	//Init Zone		
	fbSortedListMoversInQueue.ListOfMoversToCheck := THIS^.fbAssignedMovers;
	fbSortedListMoversInQueue.AccocietedTrack := THIS^.AccocietedTrack;	
	
	bInitDone := TRUE;
ELSE
	//Done
	Initialize:= S_OK;
END_IF


THIS^.fbFeedback.ActiveCommand 		:= TO_STRING(CHALET_NC.E_NcAxisCommands.Initialize);
THIS^.eActiveCommand 				:= CHALET_NC.E_NcAxisCommands.Initialize;
THIS^.fbFeedback.LastCommandAccepted:= TRUE;	
//Set done or keep in busy state	
THIS^.fbFeedback.HR := Initialize;
END_METHOD

{attribute 'monitoring':='call'}
PROPERTY MoverGapAtExit : LREAL //[mm] Every mover that leaves or passes the station gets this new gap as a target.
GET
MoverGapAtExit := fMoverGapAtExit;
END_GET
SET
IF MoverGapAtExit < XPlanarParameterlist.F_MOVER_MINIMUM_GAP_ON_TRACK THEN
	MoverGapAtExit := XPlanarParameterlist.F_MOVER_MINIMUM_GAP_ON_TRACK;
END_IF

fMoverGapAtExit := MoverGapAtExit;
END_SET
END_PROPERTY

{attribute 'monitoring':='call'}
PROPERTY MoverVelocityAtExit : LREAL //[mm/s] Every mover that leaves or passes the station gets this new velocity as a target.
GET
MoverVelocityAtExit := fMoverVelocityAtExit;
END_GET
SET
fMoverVelocityAtExit := MoverVelocityAtExit;
END_SET
END_PROPERTY

{attribute 'monitoring':='call'}
PROPERTY PositionOnTrack : LREAL
GET
PositionOnTrack := THIS^.fPositionOnTrack;
END_GET
END_PROPERTY

{attribute 'monitoring':='call'}
PROPERTY PositionOnTrackXY : REFERENCE TO PositionXY
GET
PositionOnTrackXY REF= THIS^.fbPositionOnTrackXY;
END_GET
END_PROPERTY

{attribute 'monitoring':='call'}
PROPERTY PositionXY : REFERENCE TO  PositionXY
GET
PositionXY REF= THIS^.fbPositionPlanned;
END_GET
END_PROPERTY

METHOD RegistrateStationBehinde : HRESULT
VAR_INPUT
	ipStation : I_CH_Object;
END_VAR
VAR
	ipXpStation : I_XP_Station;
END_VAR
//Check if the input implements an station interface 
IF NOT ToXpStation(ipStation,ipXpStation) THEN
	RegistrateStationBehinde := E_FAIL;
	RETURN;
END_IF

//Check if not allready is added to list
IF THIS^.fbStationsBehinde.FindObject(ipStation) THEN
	;//Allready in List
ELSE	
	THIS^.fbStationsBehinde.AddObject(ipStation);
END_IF

RegistrateStationBehinde := S_OK;
END_METHOD

METHOD SearchNextBestStationByName : ST_PathFinder_1
VAR_INPUT
	sTargedStationGroupeID : STRING;
	nPermittedSearchDepth : UINT;
	ipWhoIsAsking	: I_XP_Station;

END_VAR
VAR
	nRemainingSearchDepth 			: UINT;
	ipThisStation 					: I_XP_Station;
	ipStation 						: I_XP_Station;
	stPath							: ST_PathFinder_1;
	bIamTheAsker					: BOOL;
	bTargetFoundOnThisPath			: BOOL;
	bStationIsOnlyForDynamicChanges : BOOL;
	bStationIsFull					: BOOL;
	bStationHanMoreMoverThanAllowed : BOOL;
	bStationHasAFreePlaceInQueue 	: BOOL;
	bStationIsNotReadyToRecvMovers	: BOOL;

END_VAR
ipThisStation := (THIS^);

//Invalide input
IF ipWhoIsAsking = 0 OR sTargedStationGroupeID = '' THEN
	searchNextBestStationByName.bTargetFound := FALSE;
	searchNextBestStationByName.ipBestStation := 0;
	RETURN;
END_IF

//Has the maximum search depth been reached?
nRemainingSearchDepth := nPermittedSearchDepth - 1;
IF nRemainingSearchDepth = 0 THEN
	searchNextBestStationByName.bTargetFound := FALSE;
	searchNextBestStationByName.ipBestStation := 0;
	RETURN;
END_IF

//Is the station not aware of any other stations in front of it?
IF THIS^.fbStationsAhead.Size = 0 THEN
	searchNextBestStationByName.bTargetFound := FALSE;
	searchNextBestStationByName.ipBestStation := 0;
	RETURN;
END_IF

//Check if the requested station is this one. And not the station who is searching
IF ((THIS^.StationGroupID = sTargedStationGroupeID) AND (ipWhoIsAsking <> ipThisStation)) THEN
	stPath.bTargetFound := TRUE;
	stPath.ipBestStation := THIS^;
ELSE
	//Check the stations ahead if a movement to targed station is posible. Multiple stations incase of an switch.
	THIS^.fbStationsAhead.ResetIterator();
	WHILE THIS^.fbStationsAhead.HasNextObject() DO
		IF ToXpStation(THIS^.fbStationsAhead.GetNextObject(),ipStation) THEN
			stPath := ipStation.searchNextBestStationByName(sTargedStationGroupeID, nRemainingSearchDepth, ipWhoIsAsking);
			//the information that we are on a valid path is set if a path to destination was detected
			IF stPath.bTargetFound THEN
				bTargetFoundOnThisPath := TRUE;
			END_IF
			//if a path is found with a valid in-between position, this should be used and the finder is aborted here
			IF stPath.ipBestStation <> 0 THEN
				EXIT;
			END_IF
		END_IF
	END_WHILE
	stPath.bTargetFound := bTargetFoundOnThisPath;
END_IF

//Abort - not a valide path
IF NOT stPath.bTargetFound THEN
	searchNextBestStationByName.bTargetFound := FALSE;
	searchNextBestStationByName.ipBestStation := 0;
	RETURN;
END_IF


//evaluate whether the current best station should be overwritten by this one
bIamTheAsker					:= ipWhoIsAsking = ipThisStation;
bStationHanMoreMoverThanAllowed := (THIS^.CtsMoversInQueue > THIS^.nMoverQueueSize); //Maybe during statup if all movers are forced to station x.	
bStationIsFull					:= (THIS^.CtsEmptySpaceInQueue = 0) AND NOT (THIS^.nMoverQueueSize = 0);
bStationHasAFreePlaceInQueue 	:= (THIS^.CtsEmptySpaceInQueue > 0);
bStationIsOnlyForDynamicChanges := (THIS^.nMoverQueueSize = 0);
//bStationIsTheTarged				:= (THIS^.StationGroupID = ipMover.TargedStation);
bStationIsNotReadyToRecvMovers	:= ( NOT THIS^.bReadyToRecvMovers); 

//End of search. Return found station
IF bIamTheAsker THEN
	searchNextBestStationByName.bTargetFound := stPath.bTargetFound;
	searchNextBestStationByName.ipBestStation := stPath.ipBestStation;


//Is THIS Station a "Dynamic change station" (Queuesize = 0) and has only the purpose tho change the gap of passing movers.
//in this case, the current path should be left as it is. the station is ignored,
ELSIF bStationIsOnlyForDynamicChanges THEN
	searchNextBestStationByName.bTargetFound := stPath.bTargetFound;
	searchNextBestStationByName.ipBestStation := stPath.ipBestStation;


//This station is full, no movement posible. Do not evaluate if this station is the asker.(Dont care if my own station is full atm.)
ELSIF bStationIsFull OR bStationHanMoreMoverThanAllowed OR bStationIsNotReadyToRecvMovers OR bStationIsOnlyForDynamicChanges THEN
	searchNextBestStationByName.bTargetFound := stPath.bTargetFound;
	searchNextBestStationByName.ipBestStation := 0;

	
//This station in an valide an good targed for the mover. return this station
	ELSE
	searchNextBestStationByName.bTargetFound := TRUE;
	searchNextBestStationByName.ipBestStation := (THIS^);
END_IF
END_METHOD

{attribute 'monitoring':='call'}
PROPERTY StationGroupID : STRING
GET
StationGroupID := THIS^.sStationGroupId;
END_GET
END_PROPERTY

{attribute 'monitoring':='call'}
PROPERTY StationsAhead : I_CH_List
GET
StationsAhead := THIS^.fbStationsAhead;
END_GET
END_PROPERTY

{attribute 'monitoring':='call'}
PROPERTY StationsBehinde : I_CH_List
GET
StationsBehinde := THIS^.fbStationsBehinde;
END_GET
END_PROPERTY

{attribute 'monitoring':='call'}
PROPERTY SuppressDynamicsChange : BOOL // Suppress to change the dynamic(Gap+velocity) of passing movers. This is usefull in startup
GET
SuppressDynamicsChange := bSuppressDynamicsChange;
END_GET
SET
bSuppressDynamicsChange := SuppressDynamicsChange;
END_SET
END_PROPERTY

METHOD Update : HRESULT
VAR
	ipFirstMoverInQueue: I_XP_Mover;
	ipFirstMoverInQueuePlc : I_XP_Mover_PLC;
	ipFirstMoverInQueueObj : I_CH_Object;
	iStation: I_XP_Station;
	stPath: ST_PathFinder_1;
	bValideStationToStartMove : BOOL;
	
	ipThisStation : I_XP_Station;
END_VAR
//Force to do init befor call update
IF NOT bInitDone THEN
	THIS^.Initialize();
	RETURN;
END_IF




// ********************** Set feedback depending on active command *******************************
IF THIS^.eActiveCommand <> E_NcAxisCommands.None THEN
	fbFeedback.ActiveCommand 	:= TO_STRING(THIS^.eActiveCommand);	
END_IF

CASE THIS^.eActiveCommand OF

	E_NcAxisCommands.Initialize:
		fbFeedback.Busy 			:= NOT THIS^.bInitDone;
		fbFeedback.Done 			:= THIS^.bInitDone;
		fbFeedback.ErrorId 			:= 0;
		                        	

	ELSE//External command in subclass
		;
END_CASE


// **********************  Stop to execute commands on .done or .error ***************************
IF fbFeedback.Done OR THIS^.fbFeedback.Error THEN
	eActiveCommand 				:= E_NcAxisCommands.None;
END_IF

// Process Simulation. All functionality packed into one method for easier overwriting
THIS^.Simulation();


// If enabled start station logic
IF THIS^.ipXpSystem.Enabled THEN

	//Detect mover who is passing the station whitout be in queue. Adjust to new Gap
	IF fbTrigger.MoverDetected AND (fbTrigger.MoverAtTrigger <> 0) AND NOT THIS^.bSuppressDynamicsChange THEN
		//Only if not in this queue
		ipThisStation := (THIS^);
		IF fbTrigger.MoverAtTrigger.ParentStation <> ipThisStation THEN
			fbTrigger.MoverAtTrigger.MoveOnTrack(ipTrack	:= fbTrigger.MoverAtTrigger.LastCmdTargedTrack,
												fPosition	:= fbTrigger.MoverAtTrigger.LastCmdTargedPosition, 
												fGap		:= THIS^.fMoverGapAtExit);
		END_IF
	END_IF	
	
	//Test if the first mover is in station and send him away, if the destination is not this station
	ipFirstMoverInQueuePlc := THIS^.MoversInQueue[0];
	IF (ipFirstMoverInQueuePlc <> 0) AND_THEN (ipFirstMoverInQueuePlc.TargetStationGroupID <> THIS^.StationGroupID) AND_THEN __QUERYINTERFACE(ipFirstMoverInQueuePlc,ipFirstMoverInQueue) THEN
		//Get a path
		stPath := THIS^.searchNextBestStationByName(sTargedStationGroupeID := ipFirstMoverInQueue.TargetStationGroupID, nPermittedSearchDepth := XPlanarParameterlist.N_MAX_SEARCH_DEPTH, ipWhoIsAsking := (THIS^));
		bValideStationToStartMove := stPath.bTargetFound AND (stPath.ipBestStation <> 0);
		//Start Movement
		IF bValideStationToStartMove THEN 
			//deregister from this station and register with a new parrent station
			ipFirstMoverInQueueObj := THIS^.fbAssignedMovers.FindOID(ipFirstMoverInQueue.OID);
			THIS^.fbAssignedMovers.RemoveObject(ipFirstMoverInQueueObj);
			stPath.ipBestStation.AddMoverToQueue(ipFirstMoverInQueue);	

			//If mover is standstill in current station, send him away whit the exit gap, else use the in mover stored gap
			IF LREAL_TO_DINT(ipFirstMoverInQueue.PositionOnTrack) = LREAL_TO_DINT(THIS^.PositionOnTrack) THEN
				ipFirstMoverInQueue.MoveOnTrackToStation(ipStation := stPath.ipBestStation,
											fGap:= THIS^.fMoverGapAtExit);					
			ELSE
				ipFirstMoverInQueue.MoveOnTrackToStation(ipStation := stPath.ipBestStation,
								fGap:= ipFirstMoverInQueue.LastCmdTargedGap);
	
			END_IF	
 		END_IF     
	END_IF
END_IF



Update := S_OK;
END_METHOD

END_FUNCTION_BLOCK

// COMPONENTs/Stationen/I_XP_Station_PLC
INTERFACE I_XP_Station_PLC EXTENDS __SYSTEM.IQueryInterface

{attribute 'monitoring':='call'}
PROPERTY AreMoversInPlace : BOOL
GET
END_GET
END_PROPERTY

{attribute 'monitoring':='call'}
PROPERTY CtsEmptySpaceInQueue : UDINT
GET
END_GET
END_PROPERTY

{attribute 'monitoring':='call'}
PROPERTY CtsMoversInQueue : UDINT
GET
END_GET
END_PROPERTY

{attribute 'monitoring':='call'}
(* Return interface to mover in station. Return 0 if no mover is in station *)
PROPERTY InterfaceToMover : I_XP_Mover
GET
END_GET
END_PROPERTY

{attribute 'monitoring':='call'}
PROPERTY MoverQueueSize : UINT
GET
END_GET
SET
END_SET
END_PROPERTY

{attribute 'monitoring':='call'}
PROPERTY MoversInQueue : REFERENCE TO ARRAY [0..(CHALET_BaseComponents.BaseParameterlist.MAX_OBJECTS-1)] OF I_XP_Mover_PLC // Return a sorted list of movers in this zone. Index 0 is the mover in Front
GET
END_GET
END_PROPERTY

{attribute 'monitoring':='call'}
//prevent further movers from entering the station, 
//e.g. to prevent a collision. All movers that are already moving to reach this station will be stopped with a stop 
//and restarted with Ready True.
PROPERTY ReadyToRecvMovers : BOOL
GET
END_GET
SET
END_SET
END_PROPERTY

METHOD SendMoversToGroup : I_CH_Feedback
VAR_INPUT 
	sTargetStationGroupID : STRING;
END_VAR
END_METHOD

{attribute 'monitoring':='call'}
PROPERTY TargetPosMonitoringTime : TIME
GET
END_GET
SET
END_SET
END_PROPERTY

{attribute 'monitoring':='call'}
PROPERTY TargetPosWindow : LREAL
GET
END_GET
SET
END_SET
END_PROPERTY

{attribute 'monitoring':='call'}
PROPERTY ProcessSimulationActive : BOOL
GET
END_GET
END_PROPERTY

//If a valid time (>0seconds) is set and the configured destination station exists, then the movers will be sent away automatically after this time from now on.
METHOD SimulationMode : HRESULT
VAR_INPUT
	fProcessDuration 			: LREAL; //[s]
	sTargedStationGroupID		: STRING; //group of the targed station to automatic send after the duration
END_VAR
END_METHOD

{attribute 'monitoring':='call'}
PROPERTY AccocietedTrack : I_XP_Track
GET
END_GET
END_PROPERTY

{attribute 'monitoring':='call'}
PROPERTY Feedback : I_CH_Feedback
GET
END_GET
END_PROPERTY

{attribute 'monitoring':='call'}
PROPERTY MoverGapAtExit : LREAL //[mm] Every mover that leaves or passes the station gets this new gap as a target.
GET
END_GET
SET
END_SET
END_PROPERTY

{attribute 'monitoring':='call'}
PROPERTY PositionOnTrack : LREAL
GET
END_GET
END_PROPERTY

{attribute 'monitoring':='call'}
PROPERTY PositionOnTrackXY : REFERENCE TO PositionXY
GET
END_GET
END_PROPERTY

{attribute 'monitoring':='call'}
PROPERTY PositionXY : REFERENCE TO  PositionXY
GET
END_GET
END_PROPERTY

{attribute 'monitoring':='call'}
PROPERTY StationGroupID : STRING
GET
END_GET
END_PROPERTY

{attribute 'monitoring':='call'}
PROPERTY StationsAhead : I_CH_List
GET
END_GET
END_PROPERTY

{attribute 'monitoring':='call'}
PROPERTY StationsBehinde : I_CH_List
GET
END_GET
END_PROPERTY

END_INTERFACE

// COMPONENTs/Trigger/FB_XP_Trigger
{attribute 'no_explicit_call' := 'Do not call the body - Stick to OOP'}
FUNCTION_BLOCK FB_XP_Trigger EXTENDS FB_CH_Object IMPLEMENTS I_XP_Trigger
VAR
	{attribute 'hide'}
	bInitDone : BOOL;
	{attribute 'hide'}
	ipXpSystem : I_XP_System_Registration;
	{attribute 'hide'}
	ipAccocietedTrack : I_XP_Track;
	{attribute 'hide'}
	ipListOfMoversToCheck : CHALET_BaseComponents.I_CH_LIST;
	{attribute 'hide'}
	fTriggerPositionOnTrack : LREAL;
	{attribute 'hide'}
	eTriggerDirection : Tc3_Mc3Definitions.MC_Direction := Tc3_Mc3Definitions.MC_DIRECTION.mcDirectionPositive;
	{attribute 'hide'}
	ipMoverAtTrigger : I_XP_Mover;
	{attribute 'hide'}
	aMoversPositionLastCycle : ARRAY [0..(CHALET_BaseComponents.BaseParameterlist.MAX_OBJECTS-1)] OF LREAL; // This list is generated at the end of the PRG and contais the positions. The positions are checked in the next cycle
	{attribute 'hide'}
	aMoversTrackLastCycle : ARRAY [0..(CHALET_BaseComponents.BaseParameterlist.MAX_OBJECTS-1)] OF I_XP_Track; // This list is generated at the end of the PRG and contais the track. The tracks are checked in the next cycle
	{attribute 'hide'}
	aMoversInterfaceLastCycle : ARRAY [0..(CHALET_BaseComponents.BaseParameterlist.MAX_OBJECTS-1)] OF I_XP_Mover; // This list is generated at the end of the PRG and contais the Mover interface. The positions are checked in the next cycle
END_VAR

{attribute 'monitoring':='call'}
PROPERTY AccocietedTrack : I_XP_Track
GET
AccocietedTrack := THIS^.ipAccocietedTrack;
END_GET
SET
THIS^.ipAccocietedTrack := AccocietedTrack;
END_SET
END_PROPERTY

METHOD FB_init : BOOL
VAR_INPUT
	bInitRetains : BOOL; // if TRUE, the retain variables are initialized (warm start / cold start)
	bInCopyCode : BOOL;  // if TRUE, the instance afterwards gets moved into the copy code (online change)
	
	ipXpSystem : I_XP_System_Registration; //Interface to XTS system object
	
END_VAR
VAR_INST
	{attribute 'hide'}
	bFBInitCalledOnce : BOOL; //Do the following code once during start up and not during onlinechange
END_VAR
//Do the following code once during start up and not during onlinechange
IF NOT bFBInitCalledOnce THEN 
	;
END_IF

//Regristrate object in System if unknown
IF ipXpSystem <> 0 AND THIS^.ipXpSystem = 0 THEN
	ipXpSystem.RegisterTrigger(THIS^);
	THIS^.ipXpSystem := ipXpSystem;
END_IF

bFBInitCalledOnce := TRUE;
END_METHOD

{attribute 'monitoring':='call'}
PROPERTY HR : HRESULT
GET
IF ipAccocietedTrack <> 0 AND_THEN ipAccocietedTrack.Length > 0 THEN
	HR := S_OK;
ELSE
	HR := E_FAIL;
END_IF
END_GET
END_PROPERTY

METHOD Initialize : HRESULT
IF THIS^.ipXpSystem = 0 THEN
	//No valide interface
	Initialize := E_FAIL;
	RETURN;
END_IF

IF (THIS^.ipListOfMoversToCheck <> 0) AND (THIS^.ipAccocietedTrack <> 0) THEN
	THIS^.bInitDone := TRUE;
	Initialize := S_OK;
ELSE
	Initialize := E_FAIL;
END_IF
END_METHOD

PROPERTY ListOfMoversToCheck : I_CH_List
SET
IF ListOfMoversToCheck <> 0 THEN
	ipListOfMoversToCheck := ListOfMoversToCheck;
END_IF
END_SET
END_PROPERTY

{attribute 'monitoring':='call'}
PROPERTY MoverAtTrigger : I_XP_Mover
GET
THIS^.Prepare();//Prepare Time-critical information

MoverAtTrigger := ipMoverAtTrigger;
END_GET
END_PROPERTY

{attribute 'monitoring':='call'}
PROPERTY MoverDetected : BOOL
GET
THIS^.Prepare();//Prepare Time-critical information

MoverDetected := (ipMoverAtTrigger <> 0);
END_GET
END_PROPERTY

{attribute 'monitoring':='call'}
PROPERTY PositionOnTrack : LREAL
GET
PositionOnTrack := fTriggerPositionOnTrack;
END_GET
SET
fTriggerPositionOnTrack := PositionOnTrack;
END_SET
END_PROPERTY

(* Time-critical information is processed here, which can then be polled via the property every cycle. 
The update method is usually at the end of the program and then it is already 'outdated'. *)
METHOD PRIVATE Prepare : HRESULT
VAR
	fTrackLentgh : LREAL;
	fMoverActPos,fMoverLastPos : LREAL;
	ipMoverActTrack, ipMoverLastTrack : I_XP_Track;
	fRangePositive, fRangeNegative : LREAL;
	bTriggerIsCloseAtStartTrack, bTriggerIsCloseAtEndTrack : BOOL;
	bMoverWasInRangeNeg, bMoverWasInRangePos, bMoverIsInRangeNeg, bMoverIsInRangePos : BOOL;
	bMoverIsOnSameTrack, bMoverIsOnTrackAhead, bMoverIsOnTrackBehind, bMoverWasOnTrackAhead, bMoverWasOnTrackBehind : BOOL;
	nIdx, nIdxTrack : UDINT;
	fMaxMoveDistPerCycle : LREAL; //[mm] (2 m/s(max. xPlanar speed) * 20ms(max realistic SPS cycle time) + 10%)
END_VAR
VAR_INST
	{attribute 'hide'}
	nLastUpdatedCycleCount : UDINT;
END_VAR
VAR CONSTANT
END_VAR
//Check if this Cycle the dates are allready prepared
IF nLastUpdatedCycleCount <> TwinCAT_SystemInfoVarList._TaskInfo[THIS^.nTaskIndex].CycleCount THEN
	nLastUpdatedCycleCount := TwinCAT_SystemInfoVarList._TaskInfo[THIS^.nTaskIndex].CycleCount;
	
	//Abort on invalide interface - Get Track length
	IF ipAccocietedTrack = 0 THEN
		RETURN;
	END_IF
	fTrackLentgh := ipAccocietedTrack.Length;
	
	//Maximum distance a mover can travel in 1 plc cycle. Worstcase 2 m/s(max. xPlanar speed) * 20ms(max realistic SPS cycle time) + 10%
	fMaxMoveDistPerCycle := 2000.0(*2000mm/s=2mm/ms*) * (TwinCAT_SystemInfoVarList._TaskInfo[THIS^.nTaskIndex].CycleTime(*[100ns]*)/10_000)(*CycleTime ms*) / 1000.0 * 1.1(*10%*);
	
	//Clear last stored Mover if an new cycle has started
	THIS^.ipMoverAtTrigger := 0;
	
	//Check old list of Moverspositions and compare them to the current position of the same mover.
	//Set Trigger if the Mover pass the Station
	fRangePositive := MIN((THIS^.fTriggerPositionOnTrack + fMaxMoveDistPerCycle),fTrackLentgh);
	fRangeNegative := MAX((THIS^.fTriggerPositionOnTrack - fMaxMoveDistPerCycle),0); 
	bTriggerIsCloseAtStartTrack := (THIS^.fTriggerPositionOnTrack - fMaxMoveDistPerCycle) < 0.0;
	bTriggerIsCloseAtEndTrack 	:= (THIS^.fTriggerPositionOnTrack + fMaxMoveDistPerCycle) > fTrackLentgh;

		
	FOR nIdx := 0 TO (CHALET_BaseComponents.BaseParameterlist.MAX_OBJECTS-1) DO
		
		IF aMoversInterfaceLastCycle[nIdx] <> 0 THEN
			fMoverActPos 			:= aMoversInterfaceLastCycle[nIdx].PositionOnTrack;
			fMoverLastPos			:= aMoversPositionLastCycle[nIdx];
			ipMoverActTrack 		:= aMoversInterfaceLastCycle[nIdx].CurrentTrack;
			ipMoverLastTrack 		:= aMoversTrackLastCycle[nIdx];
			bMoverIsOnSameTrack 	:= (ipMoverActTrack = ipAccocietedTrack);
			
			//Abort if Lasttrack is not known. Example: first cycle after enabling
			IF ipMoverActTrack = 0 OR ipMoverLastTrack = 0 THEN
				RETURN;
			END_IF
			
			//Reset flags 
			bMoverIsOnTrackAhead 	:= FALSE;		bMoverIsOnTrackBehind 	:= FALSE;		bMoverWasOnTrackAhead 	:= FALSE;		bMoverWasOnTrackBehind 	:= FALSE;
			
			//Test all tracks before and after this track to recognize that the mover has just changed tracks. 
			//This is important if this trigger is near the end or beginning of a track
			FOR nIdxTrack := 0 TO (XPlanarParameterlist.N_MAX_STATIONS_AHEAD_OR_BEHIND-1) DO
				//Tracks Ahead - Mover Is/Was on Track ahead and close(cMaxMoveDistPerCycle) at beginn on track
				IF ipMoverActTrack.TracksStartFromThis[nIdxTrack] <> 0 THEN
					bMoverIsOnTrackAhead 	:= bMoverIsOnTrackAhead 	OR ((ipAccocietedTrack = ipMoverActTrack.TracksStartFromThis[nIdxTrack])  AND ((fMoverActPos - fMaxMoveDistPerCycle) < 0.0));
					bMoverWasOnTrackAhead 	:= bMoverWasOnTrackAhead 	OR ((ipAccocietedTrack = ipMoverLastTrack.TracksStartFromThis[nIdxTrack]) AND ((fMoverLastPos - fMaxMoveDistPerCycle) < 0.0));
				END_IF
				//Tracks Behind - Mover Is/Was on Track behind and close(cMaxMoveDistPerCycle) at end on track
				IF ipMoverActTrack.TracksEndAtThis[nIdxTrack] <> 0 THEN
					bMoverIsOnTrackBehind 	:= bMoverIsOnTrackBehind 	OR ((ipAccocietedTrack = ipMoverActTrack.TracksEndAtThis[nIdxTrack])  AND ((fMoverActPos	+ fMaxMoveDistPerCycle) > ipMoverActTrack.Length));
					bMoverWasOnTrackBehind 	:= bMoverWasOnTrackBehind 	OR ((ipAccocietedTrack = ipMoverLastTrack.TracksEndAtThis[nIdxTrack]) AND ((fMoverLastPos 	+ fMaxMoveDistPerCycle) > ipMoverLastTrack.Length));
				END_IF
			END_FOR
			
			//Closed track and station in close to Modulo pos
			IF bMoverIsOnSameTrack THEN
				bMoverIsOnTrackAhead 	:= ((fMoverActPos - fMaxMoveDistPerCycle) < 0.0);
				bMoverWasOnTrackAhead 	:= ((fMoverLastPos - fMaxMoveDistPerCycle) < 0.0);
				bMoverIsOnTrackBehind 	:= ((fMoverActPos	+ fMaxMoveDistPerCycle) > ipMoverActTrack.Length);
				bMoverWasOnTrackBehind 	:= ((fMoverLastPos 	+ fMaxMoveDistPerCycle) > ipMoverLastTrack.Length);
			END_IF
			
			//Check if Mover passes the station. Ex.: If the Trigger is at Pos 0mm on track, the Mover is never in bRangeNeg. For this case check for bMoverOnTrackBefore
			bMoverIsInRangePos 		:= ((fMoverActPos >= THIS^.fTriggerPositionOnTrack) AND (fMoverActPos <= fRangePositive) AND bMoverIsOnSameTrack) OR (bMoverIsOnTrackAhead 	 AND bTriggerIsCloseAtEndTrack);   
			bMoverIsInRangeNeg 		:= ((fMoverActPos <= THIS^.fTriggerPositionOnTrack) AND (fMoverActPos >= fRangeNegative) AND bMoverIsOnSameTrack) OR (bMoverIsOnTrackBehind  AND bTriggerIsCloseAtStartTrack);     
			bMoverWasInRangePos		:= ((fMoverLastPos > THIS^.fTriggerPositionOnTrack) AND (fMoverLastPos >= fRangeNegative) AND bMoverIsOnSameTrack) OR (bMoverWasOnTrackAhead  AND bTriggerIsCloseAtEndTrack);   
			bMoverWasInRangeNeg		:= ((fMoverLastPos < THIS^.fTriggerPositionOnTrack) AND (fMoverLastPos <= fRangePositive) AND bMoverIsOnSameTrack) OR (bMoverWasOnTrackBehind AND bTriggerIsCloseAtStartTrack);     			

			IF eTriggerDirection = Tc3_Mc3Definitions.MC_DIRECTION.mcDirectionPositive  AND bMoverWasInRangeNeg AND bMoverIsInRangePos AND NOT bMoverWasInRangePos THEN
				THIS^.ipMoverAtTrigger := aMoversInterfaceLastCycle[nIdx];
				RETURN;
			ELSIF eTriggerDirection = Tc3_Mc3Definitions.MC_DIRECTION.mcDirectionNegative AND bMoverIsInRangeNeg AND bMoverWasInRangePos AND NOT bMoverWasInRangeNeg THEN
				THIS^.ipMoverAtTrigger := aMoversInterfaceLastCycle[nIdx];
				RETURN;	
			END_IF
			
		END_IF
	END_FOR
END_IF
END_METHOD

{attribute 'monitoring':='call'}
PROPERTY TimeStamp : Tc2_EtherCAT.T_DCTIME64
GET
THIS^.Prepare();//Prepare Time-critical information

///zzz todo exact time stamp calculatioin
 IF ipMoverAtTrigger <> 0 THEN
	 TimeStamp := F_GetCurDcTaskTime64();
 ELSE
	 TimeStamp := 0;
 END_IF
END_GET
END_PROPERTY

{attribute 'monitoring':='call'}
PROPERTY TriggerDirection : Tc3_Mc3Definitions.MC_Direction
GET
TriggerDirection := eTriggerDirection;
END_GET
SET
IF TriggerDirection =Tc3_Mc3Definitions.MC_DIRECTION.mcDirectionPositive OR TriggerDirection = Tc3_Mc3Definitions.MC_DIRECTION.mcDirectionNegative THEN
	eTriggerDirection := TriggerDirection;
END_IF
END_SET
END_PROPERTY

METHOD Update : HRESULT
VAR
	nIndex : UINT;
	ipMover : I_XP_Mover;
END_VAR
//Force to do an init befor call update
IF NOT bInitDone THEN
	THIS^.Initialize();
	RETURN;
END_IF

//Clear array
MEMSET(destAddr:=ADR(aMoversInterfaceLastCycle),n:=SIZEOF(aMoversInterfaceLastCycle),fillByte:=0);
MEMSET(destAddr:=ADR(aMoversPositionLastCycle),n:=SIZEOF(aMoversPositionLastCycle),fillByte:=0);
MEMSET(destAddr:=ADR(aMoversTrackLastCycle),n:=SIZEOF(aMoversTrackLastCycle),fillByte:=0);

nIndex := 0;
THIS^.ipListOfMoversToCheck.ResetIterator();
WHILE THIS^.ipListOfMoversToCheck.HasNextObject() DO
	
	//Cheack all Movers fill the actposition in the array
	IF ToXpMover(THIS^.ipListOfMoversToCheck.GetNextObject(),ipMover) THEN
		aMoversInterfaceLastCycle[nIndex] 	:= ipMover;
		aMoversPositionLastCycle[nIndex] 	:= ipMover.PositionOnTrack;
		aMoversTrackLastCycle[nIndex]		:= ipMover.CurrentTrack;
		nIndex := nIndex +1;
	END_IF
	
END_WHILE
END_METHOD

END_FUNCTION_BLOCK

// COMPONENTs/Trigger/I_XP_Trigger
INTERFACE I_XP_Trigger  EXTENDS __SYSTEM.IQueryInterface

{attribute 'monitoring':='call'}
PROPERTY AccocietedTrack : I_XP_Track
GET
END_GET
SET
END_SET
END_PROPERTY

{attribute 'monitoring':='call'}
PROPERTY HR : HRESULT
GET
END_GET
END_PROPERTY

PROPERTY ListOfMoversToCheck : I_CH_List
SET
END_SET
END_PROPERTY

{attribute 'monitoring':='call'}
PROPERTY MoverAtTrigger : I_XP_Mover
GET
END_GET
END_PROPERTY

{attribute 'monitoring':='call'}
PROPERTY MoverDetected : BOOL
GET
END_GET
END_PROPERTY

{attribute 'monitoring':='call'}
PROPERTY PositionOnTrack : LREAL
GET
END_GET
SET
END_SET
END_PROPERTY

{attribute 'monitoring':='call'}
PROPERTY TimeStamp : T_DCTIME64;
GET
END_GET
END_PROPERTY

{attribute 'monitoring':='call'}
PROPERTY TriggerDirection : Tc3_Mc3Definitions.MC_Direction
GET
END_GET
SET
END_SET
END_PROPERTY

END_INTERFACE

// COMPONENTs/Zone/FB_XP_Zone
{attribute 'no_explicit_call' := 'Do not call the body - Stick to OOP'}
// Check zone start to end in positive direktion.
FUNCTION_BLOCK FB_XP_Zone EXTENDS FB_CH_Object IMPLEMENTS I_XP_Zone
VAR
	{attribute 'hide'}
	bInitDone : BOOL;
	{attribute 'hide'}
	ipXpSystem : I_XP_System_Registration; //Interface to XPlanar system 
	{attribute 'hide'}
	ipListOfMoversToCheck : CHALET_BaseComponents.I_CH_LIST;
	{attribute 'hide'}
	aMoversInZone : ARRAY [0..(CHALET_BaseComponents.BaseParameterlist.MAX_OBJECTS-1)] OF I_XP_Mover_PLC;
	{attribute 'hide'}
	fStartPositionOnTrack : LREAL;
	{attribute 'hide'}
	fEndPositionOnTrack : LREAL;	
	{attribute 'hide'}
	ipAccocietedTrack : I_XP_Track;
END_VAR

{attribute 'monitoring':='call'}
PROPERTY AccocietedTrack : I_XP_Track
GET
AccocietedTrack := THIS^.ipAccocietedTrack;
END_GET
SET
THIS^.ipAccocietedTrack := AccocietedTrack;
END_SET
END_PROPERTY

{attribute 'monitoring':='call'}
PROPERTY CtsMoversInZone : UINT
GET
VAR
	nIndex : UDINT;
END_VAR
THIS^.Prepare();//Prepare Time-critical information

//Check array for entrys, exit if fisrt empty arrayindex is found.
FOR nIndex := 0 TO (CHALET_BaseComponents.BaseParameterlist.MAX_OBJECTS-1) DO
	IF (aMoversInZone[nIndex] <> 0) THEN
		CtsMoversInZone := CtsMoversInZone +1;
	ELSE
		RETURN;
	END_IF
END_FOR
END_GET
END_PROPERTY

{attribute 'monitoring':='call'}
PROPERTY EndPositionOnTrack : LREAL
GET
EndPositionOnTrack := fEndPositionOnTrack;
END_GET
SET
fEndPositionOnTrack := EndPositionOnTrack;
END_SET
END_PROPERTY

METHOD FB_init : BOOL
VAR_INPUT
	bInitRetains : BOOL; // if TRUE, the retain variables are initialized (warm start / cold start)
	bInCopyCode : BOOL;  // if TRUE, the instance afterwards gets moved into the copy code (online change)
	
	ipXpSystem : I_XP_System_Registration; //Interface to XPlanar system object
END_VAR
VAR_INST
	{attribute 'hide'}
	bFBInitCalledOnce : BOOL; //Do the following code once during start up and not during onlinechange
END_VAR
//Do the following code once during start up and not during onlinechange
IF NOT bFBInitCalledOnce THEN 
	;
END_IF

//Regristrate object in System if unknown
IF ipXpSystem <> 0 AND THIS^.ipXpSystem = 0 THEN
	ipXpSystem.RegisterZone(THIS^);
	THIS^.ipXpSystem := ipXpSystem;
END_IF

bFBInitCalledOnce := TRUE;
END_METHOD

{attribute 'monitoring':='call'}
PROPERTY HR : HRESULT
GET
IF ipAccocietedTrack <> 0 AND_THEN ipAccocietedTrack.Length > 0 THEN
	HR := S_OK;
ELSE
	HR := E_FAIL;
END_IF
END_GET
END_PROPERTY

METHOD Initialize : HRESULT
IF THIS^.ipXpSystem = 0 THEN
	//No valide interface
	Initialize := E_FAIL;
	RETURN;
END_IF


IF (THIS^.ipListOfMoversToCheck <> 0) AND (THIS^.ipAccocietedTrack <> 0) THEN
	THIS^.bInitDone := TRUE;
	Initialize := S_OK;
ELSE
	Initialize := E_FAIL;
END_IF
END_METHOD

PROPERTY ListOfMoversToCheck : I_CH_List
SET
IF ListOfMoversToCheck <> 0 THEN
	ipListOfMoversToCheck := ListOfMoversToCheck;
END_IF
END_SET
END_PROPERTY

{attribute 'monitoring':='call'}
PROPERTY MoversInZone : REFERENCE TO ARRAY [0..(CHALET_BaseComponents.BaseParameterlist.MAX_OBJECTS-1)] OF I_XP_Mover_PLC // Return a sorted list of movers in this zone. Index 0 is the mover in Front.
GET
THIS^.Prepare();//Prepare Time-critical information

MoversInZone REF= THIS^.aMoversInZone;
END_GET
END_PROPERTY

(* Time-critical information is processed here, which can then be polled via the property every cycle. 
The update method is usually at the end of the program and then it is already 'outdated'. *)
METHOD PRIVATE Prepare : HRESULT
VAR
	nLoopIndex : UDINT;
	ipMoverPlc : I_XP_Mover_PLC;
	fDistToStart : LREAL;
	aDisanceToStart : ARRAY [0..(CHALET_BaseComponents.BaseParameterlist.MAX_OBJECTS-1)] OF LREAL;
END_VAR
VAR_INST
	{attribute 'hide'}
	nLastUpdatedCycleCount : UDINT;
END_VAR
//Check if this Cycle the dates are allready prepared
IF nLastUpdatedCycleCount <> TwinCAT_SystemInfoVarList._TaskInfo[THIS^.nTaskIndex].CycleCount THEN
	nLastUpdatedCycleCount := TwinCAT_SystemInfoVarList._TaskInfo[THIS^.nTaskIndex].CycleCount;

	//Clear array
	MEMSET(destAddr:=ADR(aMoversInZone),n:=SIZEOF(aMoversInZone),fillByte:=0);
	
	//Cheack all Movers and generate a sorted list of all mover in this zone
	THIS^.ipListOfMoversToCheck.ResetIterator();
	WHILE THIS^.ipListOfMoversToCheck.HasNextObject() DO
		IF __QUERYINTERFACE(THIS^.ipListOfMoversToCheck.GetNextObject(),ipMoverPlc) THEN
			
			//If in zone
			IF ipMoverPlc.CurrentTrack = THIS^.ipAccocietedTrack AND_THEN (fStartPositionOnTrack <= ipMoverPlc.PositionOnTrack) AND (fEndPositionOnTrack >= ipMoverPlc.PositionOnTrack) AND (fStartPositionOnTrack <= fEndPositionOnTrack) THEN
				fDistToStart := fEndPositionOnTrack - ipMoverPlc.PositionOnTrack;
				
				//Check array of movers and decide if the current one is closer to 
				FOR nLoopIndex := 0 TO (CHALET_BaseComponents.BaseParameterlist.MAX_OBJECTS-1) DO
					//empty array position
					IF aMoversInZone[nLoopIndex] = 0 THEN
						aMoversInZone[nLoopIndex] := ipMoverPlc;
						aDisanceToStart[nLoopIndex] := fDistToStart;
						EXIT;
						
					//Closer Mover found, move whole array 	
					ELSIF aDisanceToStart[nLoopIndex] > fDistToStart THEN
						MEMMOVE(srcAddr := ADR(aMoversInZone[nLoopIndex]), destAddr := ADR(aMoversInZone[nLoopIndex+1]), n := (SIZEOF(aMoversInZone[0])*(CHALET_BaseComponents.BaseParameterlist.MAX_OBJECTS-1)));
						MEMMOVE(srcAddr := ADR(aDisanceToStart[nLoopIndex]), destAddr := ADR(aDisanceToStart[nLoopIndex+1]), n := (SIZEOF(aDisanceToStart[0])*(CHALET_BaseComponents.BaseParameterlist.MAX_OBJECTS-1)));
						aMoversInZone[nLoopIndex] := ipMoverPlc;
						aDisanceToStart[nLoopIndex] := fDistToStart;
						EXIT;
						
					//check next position	
					ELSE 
						;
					END_IF
				END_FOR
			END_IF
		END_IF
	END_WHILE
END_IF
END_METHOD

{attribute 'monitoring':='call'}
PROPERTY StartPositionOnTrack : LREAL
GET
StartPositionOnTrack := fStartPositionOnTrack;
END_GET
SET
fStartPositionOnTrack := StartPositionOnTrack;
END_SET
END_PROPERTY

METHOD Update : HRESULT
VAR

END_VAR
// Nothing todo in Update. Check Prepare
END_METHOD

END_FUNCTION_BLOCK

// COMPONENTs/Zone/I_XP_Zone
INTERFACE I_XP_Zone

{attribute 'monitoring':='call'}
PROPERTY AccocietedTrack : I_XP_Track
GET
END_GET
SET
END_SET
END_PROPERTY

{attribute 'monitoring':='call'}
PROPERTY CtsMoversInZone : UINT
GET
END_GET
END_PROPERTY

{attribute 'monitoring':='call'}
PROPERTY EndPositionOnTrack : LREAL
GET
END_GET
SET
END_SET
END_PROPERTY

{attribute 'monitoring':='call'}
PROPERTY HR : HRESULT
GET
END_GET
END_PROPERTY

PROPERTY ListOfMoversToCheck : I_CH_List
SET
END_SET
END_PROPERTY

{attribute 'monitoring':='call'}
PROPERTY MoversInZone : REFERENCE TO ARRAY [0..(CHALET_BaseComponents.BaseParameterlist.MAX_OBJECTS-1)] OF I_XP_Mover_PLC // Return a sorted list of movers in this zone. Index 0 is the mover in Front.
GET
END_GET
END_PROPERTY

{attribute 'monitoring':='call'}
PROPERTY StartPositionOnTrack : LREAL
GET
END_GET
SET
END_SET
END_PROPERTY

END_INTERFACE

// COMPONENTs/System/I_XP_System_PLC
INTERFACE I_XP_System_PLC EXTENDS I_CH_Object

METHOD Disable : I_CH_Feedback
VAR_INPUT
END_VAR
END_METHOD

{attribute 'monitoring':='call'}
PROPERTY Disabled : BOOL
GET
END_GET
END_PROPERTY

METHOD Enable : I_CH_Feedback
VAR_INPUT
END_VAR
END_METHOD

{attribute 'monitoring':='call'}
PROPERTY Enabled : BOOL
GET
END_GET
END_PROPERTY

{attribute 'monitoring':='call'}
PROPERTY Enviroment : I_XP_Environment
GET
END_GET
END_PROPERTY

{attribute 'monitoring':='call'}
PROPERTY Feedback : CHALET_BaseComponents.I_CH_Feedback
GET
END_GET
END_PROPERTY

METHOD Initialize : HRESULT
VAR_INPUT
END_VAR
END_METHOD

{attribute 'monitoring':='call'}
PROPERTY Initialized : BOOL
GET
END_GET
END_PROPERTY

{attribute 'monitoring':='call'}
PROPERTY Movers : CHALET_BaseComponents.I_CH_LIST
GET
END_GET
END_PROPERTY

METHOD Station : I_XP_Station_PLC
VAR_INPUT
	sLUID : STRING;
END_VAR
END_METHOD

{attribute 'monitoring':='call'}
PROPERTY Stations : CHALET_BaseComponents.I_CH_LIST
GET
END_GET
END_PROPERTY

{attribute 'monitoring':='call'}
PROPERTY Tracks : CHALET_BaseComponents.I_CH_LIST
GET
END_GET
END_PROPERTY

{attribute 'monitoring':='call'}
PROPERTY Triggers : CHALET_BaseComponents.I_CH_LIST
GET
END_GET
END_PROPERTY

METHOD Update : HRESULT
VAR_INPUT
END_VAR
END_METHOD

METHOD ValideStationGroupID : BOOL //Return TRUE if group is existing
VAR_INPUT
	sStationGroupID	: STRING; //Group of the targed station
END_VAR
END_METHOD

//Return TRUE if unique station id is valid. if false, interfacepointer is zero -> fatal error
METHOD ValidLUID : BOOL
VAR_INPUT
	sLUID : STRING;
END_VAR
END_METHOD

{attribute 'monitoring':='call'}
PROPERTY Zones : CHALET_BaseComponents.I_CH_LIST
GET
END_GET
END_PROPERTY

END_INTERFACE

// COMPONENTs/System/FB_XP_System
{attribute 'no_explicit_call' := 'Do not call the body - Stick to OOP'}
(* XPlanar System - 1 per associated XPlanar 
	The system is the container and organizer for all subsequent XPlanar objects. All objects are registered with this system*)
FUNCTION_BLOCK FB_XP_System EXTENDS FB_CH_Object IMPLEMENTS I_XP_System_Registration, I_XP_System_PLC
VAR	
	{attribute 'hide'}
	bInitDone : BOOL;
	bErrorDuringFbInit : BOOL; // Not possible to reset
	{attribute 'hide'}                   	
	eActiveCommand 		: CHALET_Nc.E_NcAxisCommands := CHALET_Nc.E_NcAxisCommands.None;
	{attribute 'hide'}
    fbMovers     : FB_CH_List;
	{attribute 'hide'}	
    fbTracks     : FB_CH_List;
	{attribute 'hide'}	
	fbStations 	 : FB_CH_List;
	{attribute 'hide'}	
	fbTriggers 	 : FB_CH_List;
	{attribute 'hide'}	
	fbZones 	 : FB_CH_List;
	{attribute 'hide'}	
    ipGroup       : I_XP_Group;
	{attribute 'hide'}	
    ipEnvironment : I_XP_Environment;
	{attribute 'hide'}
    nSeqEnabling  : UINT;
	{attribute 'hide'}
	nSeqJoiningTrack : UINT;
	{attribute 'hide'}
	nSeqJoiningStation : UINT;
	{attribute 'hide'}	
    nSeqDisabling  : UINT := SEQ_DONE;
	{attribute 'hide'}
	fbFeedback : FB_CH_Feedback;
END_VAR
VAR CONSTANT
	{attribute 'hide'}
	SEQ_DONE : UINT := 999;
END_VAR

METHOD PROTECTED JoiningStation : HRESULT
VAR
	hr : HRESULT;
	ipEachMover : I_XP_Mover;
	ipEachMoverPlc : I_XP_Mover_PLC;
	ipEachMoverInStation : I_XP_Mover;
	ipEachStation : I_XP_Station;
	ipFirstStation : I_XP_Station;
	ipParentStation : I_XP_Station;
	ipTempMoverPlc : I_XP_Mover_PLC;
	
	//during move on track
	fVelo, fAccDec	: Tc3_Mc3Definitions.MC_LREAL := Tc3_Mc3Definitions.MC_DEFAULT;
END_VAR
VAR_INST
	{attribute 'hide'}	
	fbDelayJoiningStation : TON;
END_VAR
CASE nSeqJoiningStation OF

	0: //Init
		fbDelayJoiningStation.IN := FALSE;
		nSeqJoiningStation := 10;
	
		
	10:	//Distribute the movers to the available stations.
		(*Send the movers to the last assigned station:
		  For this purpose, the list of assigned movers is checked at each station and the mover is given a new move command to the station.
		  If there are still movers in the system that do not have a move command, these are sent to station 1. Typically after starting up
		  *)
		
		//Do for each mover in a station
		THIS^.fbStations.ResetIterator();    
		WHILE THIS^.fbStations.HasNextObject() DO
			ToXpStation(THIS^.fbStations.GetNextObject(),ipEachStation);
				//Do for all in station assigned Movers
				ipEachStation.AssignedMovers.ResetIterator();
				WHILE ipEachStation.AssignedMovers.HasNextObject() DO
					ToXpMover(ipEachStation.AssignedMovers.GetNextObject(),ipEachMoverInStation);
					//Send to assigned station - Shortest way
					hr := GetMostSignificant(hr, ipEachMoverInStation.MoveOnTrack_ShortestWay(ipTrack	:= ipEachStation.AccocietedTrack, 
																							  fPosition	:= ipEachStation.PositionOnTrack,
																							  fGap 		:= ipEachMoverInStation.LastCmdTargedGap));
				END_WHILE
		END_WHILE        
		nSeqJoiningStation := 20;
		
	20:	//Test if there is an Mover whitout an active TargedStation (first startup)
		//Send them to first station
		THIS^.fbStations.ResetIterator();
		IF THIS^.fbStations.HasNextObject() THEN
			//Get interface to first Station in list
			ToXpStation(THIS^.fbStations.GetNextObject(),ipFirstStation);
			//Set as targed station the first station in list. but as the parent the station in front of the first one(if existing) 
			//(the parent station is not necessarily the target station. But the station that is responsible for sending the mover forward if necessary)
			ipFirstStation.StationsAhead.ResetIterator();
			ToXpStation(ipFirstStation.StationsAhead.GetNextObject(),ipParentStation);
			
			//Check for mover whitout a targed station
			THIS^.fbMovers.ResetIterator();
			WHILE THIS^.fbMovers.HasNextObject() DO
				//Do for all Movers whitout a targed station
				IF ToXpMover(THIS^.fbMovers.GetNextObject(),ipEachMover) AND_THEN (ipEachMover.TargetStationGroupID = '') AND_THEN __QUERYINTERFACE(ipEachMover,ipEachMoverPlc) THEN
					//Set Path dynamic constraint to settings in XPlanarParameterlist. 0=Defalt
					IF XPlanarParameterlist.F_ENABLING_ON_TRACK_VELOCITY <> 0 THEN fVelo := XPlanarParameterlist.F_ENABLING_ON_TRACK_VELOCITY;END_IF
					IF XPlanarParameterlist.F_ENABLING_ON_TRACK_ACC_DEC <> 0 THEN fAccDec := XPlanarParameterlist.F_ENABLING_ON_TRACK_ACC_DEC;END_IF
				
					//Increase or decrease the mover DynConstraint for approaching the station 
					ipEachMoverPlc.SetDynConstraint_Path(	V:= fVelo, 
															A:= fAccDec, 
															D:= fAccDec, 
															J:= Tc3_Mc3Definitions.MC_DEFAULT);
		
					//Set as targed station the first station in list. but as the parent the station in front of the first one(if existing) 
					IF ipParentStation <> 0 THEN
						hr := GetMostSignificant(hr, ipEachMover.MoveOnTrackToStation(ipParentStation, XPlanarParameterlist.F_GAP_STARTUP));
						hr := GetMostSignificant(hr, ipParentStation.AddMoverToQueue(ipEachMover));
						ipEachMover.TargetStationGroupID := ipFirstStation.StationGroupID;
					ELSE
						//If no partent station is existing
						hr := GetMostSignificant(hr, ipEachMover.MoveOnTrackToStation(ipFirstStation, XPlanarParameterlist.F_GAP_STARTUP));
						hr := GetMostSignificant(hr, ipFirstStation.AddMoverToQueue(ipEachMover));
						ipEachMover.TargetStationGroupID := ipFirstStation.StationGroupID;
					END_IF
					
					
					//Set Path dynamic constraint back to default
					ipEachMoverPlc.SetDynConstraint_Path(	V:= Tc3_Mc3Definitions.MC_DEFAULT, 
															A:= Tc3_Mc3Definitions.MC_DEFAULT, 
															D:= Tc3_Mc3Definitions.MC_DEFAULT, 
															J:= Tc3_Mc3Definitions.MC_DEFAULT);
		
				END_IF
			END_WHILE
		END_IF

		nSeqJoiningStation := 30;
		
	30: //Delay to allow the movers to start movement
		fbDelayJoiningStation.IN := TRUE;
		fbDelayJoiningStation.PT := T#2S;
		IF fbDelayJoiningStation.Q THEN
			nSeqJoiningStation := 40;
			fbDelayJoiningStation.IN := FALSE;
		END_IF
	
	
	40: //Wait for all movers until the movement is completed(speed =0)
		THIS^.fbMovers.ResetIterator();
		WHILE THIS^.fbMovers.HasNextObject() DO
			IF ToXpMover(THIS^.fbMovers.GetNextObject(),ipEachMover) THEN
				//Check all movers if an error is active
				IF ipEachMover.Feedback.Error THEN
					hr := GetMostSignificant(hr, ipEachMover.Feedback.HR);
				//Wait for all movers to stop/finish movement
				ELSIF NOT (ipEachMover.PlanarMover.MCTOPLC.SETONTRACK.SetVelo = 0.0) THEN
					hr := GetMostSignificant(hr, S_PENDING);
				END_IF
			END_IF
		END_WHILE
		
		IF CheckOk(hr) THEN 
			nSeqJoiningStation := SEQ_DONE;
		ELSIF FAILED(hr) THEN
			nSeqJoiningStation := 1000 + nSeqJoiningStation;
		END_IF			

	
	1000..1999://Error
		hr := GetMostSignificant(hr, E_FAIL);
END_CASE

//Update
fbDelayJoiningStation();


//Return value
IF FAILED(hr) THEN 
	//Error
    JoiningStation := GetMostSignificant(hr, E_FAIL);
ELSIF (nSeqJoiningStation = SEQ_DONE) THEN
	//Done
    JoiningStation := S_OK;
ELSE
	//Busy
    JoiningStation := S_PENDING;;
END_IF
END_METHOD

METHOD PROTECTED JoiningTrack : HRESULT
VAR	
	hr : HRESULT;
	ipClosestTrack : I_XP_Track;	
	ipEachMover : I_XP_Mover;
	ipEachTrack : I_XP_Track;
	fDistance : LREAL;
	fShortestDistance : LREAL;
END_VAR
CASE nSeqJoiningTrack OF

	0: //Init
		nSeqJoiningTrack := 10;
	
		
	
	10:// Join closest track
		THIS^.fbMovers.ResetIterator();
		WHILE THIS^.fbMovers.HasNextObject() DO
			IF ToXpMover(THIS^.fbMovers.GetNextObject(),ipEachMover) THEN
				
				//check all track to decide which is the closest
				THIS^.fbTracks.ResetIterator();
				//start with the greatest possible distance, so that each track is definitely closer
				fShortestDistance := CHALET_BaseComponents.GVL_Datatypes.cMaxLreal; 
				WHILE THIS^.fbTracks.HasNextObject() DO
					IF ToXpTrack(THIS^.fbTracks.GetNextObject(),ipEachTrack) THEN
						fDistance := ipEachMover.DistToTrack(ipEachTrack);
						//closer track found
						IF fDistance <= fShortestDistance THEN
							ipClosestTrack := ipEachTrack;
							fShortestDistance := fDistance;
						END_IF
					END_IF
				END_WHILE
				
				//send mover to found closest track
				IF ipClosestTrack <> 0 THEN
					hr := GetMostSignificant(hr, ipEachMover.JoinTrack(ipClosestTrack));
				ELSE
					hr := GetMostSignificant(hr, E_FAIL);
				END_IF
			END_IF
		END_WHILE
		nSeqJoiningTrack := 20;
		
		
	20: // Joining closest track check feedback
		IF NOT fbTracks.IsEmpty THEN
			THIS^.fbMovers.ResetIterator();
			WHILE THIS^.fbMovers.HasNextObject() DO
				IF ToXpMover(THIS^.fbMovers.GetNextObject(),ipEachMover) THEN
					
					// Check mover errors
					hr := GetMostSignificant(hr, ipEachMover.Feedback.HR);
					
					//Check if Mover is on track
					IF NOT (ipEachMover.Mode = MC_PLANAR_MOVER_COMMAND_MODE.OnTrack) THEN
						hr := GetMostSignificant(hr, S_PENDING);
					END_IF
				END_IF
			END_WHILE
		END_IF
		
		IF CheckOk(hr) THEN 
			nSeqJoiningTrack := SEQ_DONE;
		ELSIF FAILED(hr) THEN
			nSeqJoiningTrack := 1000 + nSeqJoiningTrack;
		END_IF			

		
	1000..1999://Error
		hr := GetMostSignificant(hr, E_FAIL);
END_CASE

		
		
//Return value
IF FAILED(hr) THEN 
	//Error
    JoiningTrack := GetMostSignificant(hr, E_FAIL);
ELSIF (nSeqJoiningTrack = SEQ_DONE) THEN
	//Done
    JoiningTrack := S_OK;
ELSE
	//Busy
    JoiningTrack := S_PENDING;;
END_IF
END_METHOD

METHOD Disable : I_CH_Feedback
VAR_INPUT
END_VAR
//Disable is allways posible

THIS^.nSeqDisabling 	:= 1;
THIS^.nSeqEnabling 	:= 0;

THIS^.eActiveCommand 				:= CHALET_NC.E_NcAxisCommands.Disable;
THIS^.fbFeedback.LastCommandAccepted:= TRUE;		
THIS^.fbFeedback.Busy 				:= TRUE;
		
Disable := THIS^.fbFeedback;
END_METHOD

{attribute 'monitoring':='call'}
PROPERTY Disabled : BOOL
GET
Disabled := nSeqDisabling = SEQ_DONE
									OR (nSeqDisabling = 0 AND nSeqEnabling = 0);
END_GET
END_PROPERTY

METHOD PROTECTED Disabling : HRESULT
VAR
	hr : HRESULT;
	bOk : BOOL := TRUE;
	iTempMover : I_XP_Mover;
	iTempTrack : I_XP_Track;
END_VAR
Disabling := S_PENDING;
CASE nSeqDisabling OF
	0: // Idle
		Disabling := S_OK;
		
		
	1: // Halt movers
		THIS^.fbMovers.ResetIterator();
		WHILE THIS^.fbMovers.HasNextObject() DO
			IF ToXpMover(THIS^.fbMovers.GetNextObject(),iTempMover) THEN
				hr := GetMostSignificant(hr, iTempMover.Halt());
			END_IF
		END_WHILE
		
		IF CheckOk(hr) THEN 
			nSeqDisabling := 20;
		ELSE
			nSeqDisabling := 1000 + nSeqDisabling;
		END_IF	
	
		
	20: // Halting movers
		THIS^.fbMovers.ResetIterator();
		WHILE THIS^.fbMovers.HasNextObject() DO
			IF ToXpMover(THIS^.fbMovers.GetNextObject(),iTempMover) THEN
				bOk := bOk AND iTempMover.PlanarMover.MCTOPLC.SET.SetVelo.x = 0;
				bOk := bOk AND iTempMover.PlanarMover.MCTOPLC.SET.SetVelo.y = 0;
				bOk := bOk AND iTempMover.PlanarMover.MCTOPLC.SET.SetVelo.z = 0;
				bOk := bOk AND iTempMover.PlanarMover.MCTOPLC.SET.SetVelo.a = 0;
				bOk := bOk AND iTempMover.PlanarMover.MCTOPLC.SET.SetVelo.b = 0;
				bOk := bOk AND iTempMover.PlanarMover.MCTOPLC.SET.SetVelo.c = 0;
			END_IF
		END_WHILE
		
		IF bOk THEN 
			nSeqDisabling := 30;
		END_IF	
		
	
	30: // Reset movers
		THIS^.fbMovers.ResetIterator();
		WHILE THIS^.fbMovers.HasNextObject() DO
			IF ToXpMover(THIS^.fbMovers.GetNextObject(),iTempMover) THEN
				hr := GetMostSignificant(hr, iTempMover.Reset());
			END_IF
		END_WHILE
		
		IF CheckOk(hr) THEN 
			nSeqDisabling := 40;
		ELSE
			nSeqDisabling := 1000 + nSeqDisabling;
		END_IF		
		
		
	40: // Resetting movers
		THIS^.fbMovers.ResetIterator();
		WHILE THIS^.fbMovers.HasNextObject() DO
			IF ToXpMover(THIS^.fbMovers.GetNextObject(),iTempMover) THEN
				hr := GetMostSignificant(hr, iTempMover.Feedback.HR);
			END_IF
		END_WHILE
		
		IF CheckOk(hr) THEN 
			nSeqDisabling := 50;
		ELSIF FAILED(hr) THEN
			nSeqDisabling := 1000 + nSeqDisabling;
		END_IF
		
		
	50: // Disable movers
		THIS^.fbMovers.ResetIterator();
		WHILE THIS^.fbMovers.HasNextObject() DO
			IF ToXpMover(THIS^.fbMovers.GetNextObject(),iTempMover) THEN
				hr := GetMostSignificant(hr, iTempMover.Disable());
			END_IF
		END_WHILE
		
		IF CheckOk(hr) THEN 
			nSeqDisabling := 60;
		ELSE
			nSeqDisabling := 1000 + nSeqDisabling;
		END_IF			
		
		
	60: // Disabling movers
		THIS^.fbMovers.ResetIterator();
		WHILE THIS^.fbMovers.HasNextObject() DO
			IF ToXpMover(THIS^.fbMovers.GetNextObject(),iTempMover) THEN
				hr := GetMostSignificant(hr, iTempMover.Feedback.HR);
			END_IF
		END_WHILE
		
		IF CheckOk(hr) THEN 
			nSeqDisabling := 61;
		ELSIF FAILED(hr) THEN
			nSeqDisabling := 1000 + nSeqDisabling;
		END_IF		


	61: // Reset track
		THIS^.fbTracks.ResetIterator();
		WHILE THIS^.fbTracks.HasNextObject() DO
			IF ToXpTrack(THIS^.fbTracks.GetNextObject(),iTempTrack) THEN
				hr := GetMostSignificant(hr, iTempTrack.Reset());
			END_IF
		END_WHILE
		
		IF CheckOk(hr) THEN 
			nSeqDisabling := 62;
		ELSE
			nSeqDisabling := 1000 + nSeqDisabling;
		END_IF		
		
		
	62: // Resetting track
		THIS^.fbTracks.ResetIterator();
		WHILE THIS^.fbTracks.HasNextObject() DO
			IF ToXpTrack(THIS^.fbTracks.GetNextObject(),iTempTrack) THEN
				hr := GetMostSignificant(hr, iTempTrack.Feedback.HR);
			END_IF
		END_WHILE
		
		IF CheckOk(hr) THEN 
			nSeqDisabling := 63;
		ELSIF FAILED(hr) THEN
			nSeqDisabling := 1000 + nSeqDisabling;
		END_IF	

				
	63: // Reset group
		hr := ipGroup.Reset();
		
		IF CheckOk(hr) THEN 
			nSeqDisabling := 64;
		ELSE
			nSeqDisabling := 1000 + nSeqDisabling;
		END_IF		
		
		
	64: // Resetting group
		hr := ipGroup.Feedback.HR;
		
		IF CheckOk(hr) THEN 
			nSeqDisabling := 70;
		ELSIF FAILED(hr) THEN
			nSeqDisabling := 1000 + nSeqDisabling;
		END_IF		
		
		
		

   70: // Disable tracks
		THIS^.fbTracks.ResetIterator();
		WHILE THIS^.fbTracks.HasNextObject() DO
			IF ToXpTrack(THIS^.fbTracks.GetNextObject(),iTempTrack) THEN
				hr := GetMostSignificant(hr, iTempTrack.Disable());
			END_IF
		END_WHILE
		
		IF CheckOk(hr) THEN 
			nSeqDisabling := 80;
		ELSE
			nSeqDisabling := 1000 + nSeqDisabling;
		END_IF			
   
		
   80: // Disabling tracks
		THIS^.fbTracks.ResetIterator();
		WHILE THIS^.fbTracks.HasNextObject() DO
			IF ToXpTrack(THIS^.fbTracks.GetNextObject(),iTempTrack) THEN
				hr := GetMostSignificant(hr, iTempTrack.Feedback.HR);
			END_IF
		END_WHILE
		
		IF CheckOk(hr) THEN 
			nSeqDisabling := 90;
		ELSIF FAILED(hr) THEN
			nSeqDisabling := 1000 + nSeqDisabling;
		END_IF	
				

	90: // Disable group
		hr := ipGroup.Disable();
		
		IF CheckOk(hr) THEN 
			nSeqDisabling := 100;
		ELSE
			nSeqDisabling := 1000 + nSeqDisabling;
		END_IF	
		
		
   100: // Disabling group
		hr := ipGroup.Feedback.HR;
		
		IF CheckOk(hr) THEN 
			nSeqDisabling := 105;
		ELSIF FAILED(hr) THEN
			nSeqDisabling := 1000 + nSeqDisabling;
		END_IF	

		
  105: // Remove tracks from group
		THIS^.fbTracks.ResetIterator();
		WHILE THIS^.fbTracks.HasNextObject() DO
			IF ToXpTrack(THIS^.fbTracks.GetNextObject(),iTempTrack) THEN
				hr := GetMostSignificant(hr, iTempTrack.RemoveFromGroup());
			END_IF
		END_WHILE
		
		IF CheckOk(hr) THEN 
			nSeqDisabling := 106;
		ELSE
			nSeqDisabling := 1000 + nSeqDisabling;
		END_IF			
   
		
   106: // Removing tracks from group
		THIS^.fbTracks.ResetIterator();
		WHILE THIS^.fbTracks.HasNextObject() DO
			IF ToXpTrack(THIS^.fbTracks.GetNextObject(),iTempTrack) THEN
				bOk := bOk AND iTempTrack.PlanarTrack.MCTOPLC_STD.GroupOID = 0;
			END_IF
		END_WHILE
		
		IF bOk THEN 
			nSeqDisabling := 110;
		END_IF	
		
		
	110: // Remove movers from group
		THIS^.fbMovers.ResetIterator();
		WHILE THIS^.fbMovers.HasNextObject() DO
			IF ToXpMover(THIS^.fbMovers.GetNextObject(),iTempMover) THEN
				hr := GetMostSignificant(hr, iTempMover.RemoveFromGroup());
			END_IF
		END_WHILE
		
		IF CheckOk(hr) THEN 
			nSeqDisabling := 120;
		ELSE
			nSeqDisabling := 1000 + nSeqDisabling;
		END_IF		
	
		
	120: // Removing movers from group
		THIS^.fbMovers.ResetIterator();
		WHILE THIS^.fbMovers.HasNextObject() DO
			IF ToXpMover(THIS^.fbMovers.GetNextObject(),iTempMover) THEN
				bOk := bOk AND iTempMover.PlanarMover.MCTOPLC.STD.GroupOID = 0;
			END_IF
		END_WHILE
		
		IF bOk THEN 
			nSeqDisabling := 130;
		END_IF		
	
		
	130: // Remove envirement from group
		hr := ipEnvironment.RemoveFromGroup();
		
		IF CheckOk(hr) THEN 
			nSeqDisabling := 140;
		ELSE
			nSeqDisabling := 1000 + nSeqDisabling;
		END_IF		
		
		
   140: // Removing envirement from group
		//IF CheckOk(iEnvironment.HR) OR (iEnvironment.Self.MCTOPLC_STD.GroupOID = 0) THEN 
		hr := ipEnvironment.Feedback.HR;
	
		IF CheckOk(hr) THEN 
			nSeqDisabling := SEQ_DONE;
		ELSIF FAILED(hr) THEN
			nSeqDisabling := 1000 + nSeqDisabling;
		END_IF	
		
	
   SEQ_DONE: //Done
   		Disabling := S_OK;

		
	1000..1999://Error
		hr := GetMostSignificant(hr, E_FAIL);

END_CASE

// Propagate error
IF FAILED(hr) THEN
	Disabling := hr;
END_IF
END_METHOD

METHOD Enable : I_CH_Feedback
VAR_INPUT
END_VAR
IF NOT THIS^.fbFeedback.Done THEN
	//Error active/not ready
	THIS^.fbFeedback.LastCommandAccepted 	:= FALSE;

ELSIF nSeqEnabling <> 0 THEN
	//System is partial or full enabled. Disable first.
	THIS^.fbFeedback.LastCommandAccepted 	:= FALSE;
ELSE
	THIS^.nSeqDisabling 	:= 0;
	THIS^.nSeqEnabling 	:= 1;
	
	THIS^.eActiveCommand 				:= CHALET_NC.E_NcAxisCommands.Enable;
	THIS^.fbFeedback.LastCommandAccepted:= TRUE;		
	THIS^.fbFeedback.Busy 				:= TRUE;	
END_IF

Enable := THIS^.fbFeedback;
END_METHOD

{attribute 'monitoring':='call'}
PROPERTY Enabled : BOOL
GET
Enabled := nSeqEnabling = SEQ_DONE;
END_GET
END_PROPERTY

METHOD PROTECTED Enabling : HRESULT
VAR
	hr : HRESULT;
	
	ipTempMover : I_XP_Mover;
	ipTempMoverPlc : I_XP_Mover_PLC;
	ipTempStation : I_XP_Station;
	ipTempTrack : I_XP_Track;
	
	lrCRotationShortestPos : LREAL;
END_VAR

VAR_INST
	fbTimeOutSeq : TON; 
	nlastState : UINT;
END_VAR
Enabling := S_PENDING;
CASE nSeqEnabling OF
	0: // Idle
		Enabling := S_OK;	
		
	1: //Redetect all movers on real system
		IF THIS^.ipEnvironment.UtilityEnvirement.XpuTcIo(1).GetOperationMode() = OperationMode.Normal THEN
			THIS^.ipEnvironment.UtilityEnvirement.XpuTcIo(1).SetStartMoverRedetection();	
		END_IF
		nSeqEnabling := 5;

		
	5: //Compare detectet and expectet movers	
	   //timeout is monitored in this sequence
		IF (THIS^.ipEnvironment.UtilityEnvirement.XpuTcIo(1).GetMoverDetectionInfos().APM4220Detected = THIS^.ipEnvironment.UtilityEnvirement.XpuTcIo(1).GetMoverDetectionInfos().APM4220Expected AND
			THIS^.ipEnvironment.UtilityEnvirement.XpuTcIo(1).GetMoverDetectionInfos().APM4221Detected = THIS^.ipEnvironment.UtilityEnvirement.XpuTcIo(1).GetMoverDetectionInfos().APM4221Expected AND
			THIS^.ipEnvironment.UtilityEnvirement.XpuTcIo(1).GetMoverDetectionInfos().APM4330Detected = THIS^.ipEnvironment.UtilityEnvirement.XpuTcIo(1).GetMoverDetectionInfos().APM4330Expected AND
			THIS^.ipEnvironment.UtilityEnvirement.XpuTcIo(1).GetMoverDetectionInfos().APM4550Detected = THIS^.ipEnvironment.UtilityEnvirement.XpuTcIo(1).GetMoverDetectionInfos().APM4550Expected AND
			THIS^.ipEnvironment.UtilityEnvirement.XpuTcIo(1).GetMoverDetectionInfos().TotalDetected   = THIS^.ipEnvironment.UtilityEnvirement.XpuTcIo(1).GetMoverDetectionInfos().TotalExpected 	
		   )THEN
			nSeqEnabling := 20;
		END_IF	
			
		
		
	20: // Reset movers
		THIS^.fbMovers.ResetIterator();
		WHILE THIS^.fbMovers.HasNextObject() DO
			IF ToXpMover(THIS^.fbMovers.GetNextObject(),ipTempMover) THEN
				hr := GetMostSignificant(hr, ipTempMover.Reset());
			END_IF
		END_WHILE
		
		IF CheckOk(hr) THEN 
			nSeqEnabling := 21;
		ELSE
			nSeqEnabling := 1000 + nSeqEnabling;
		END_IF		
			
	21: // Resetting movers
		THIS^.fbMovers.ResetIterator();
		WHILE THIS^.fbMovers.HasNextObject() DO
			IF ToXpMover(THIS^.fbMovers.GetNextObject(),ipTempMover) THEN
				hr := GetMostSignificant(hr, ipTempMover.Feedback.HR);
			END_IF
		END_WHILE
		
		IF CheckOk(hr) THEN 
			nSeqEnabling := 30;
		ELSIF FAILED(hr) THEN
			nSeqEnabling := 1000 + nSeqEnabling;
		END_IF

		
		
	30: // Configure environment
		hr := ipEnvironment.Configure();
		
		IF CheckOk(hr) THEN 
			nSeqEnabling := 31;
		ELSE
			nSeqEnabling := 1000 + nSeqEnabling;
		END_IF	

	31: // Configuring environment
		hr := ipEnvironment.Feedback.HR;
		
		IF CheckOk(hr) THEN 
			nSeqEnabling := 50;
		ELSIF FAILED(hr) THEN
			nSeqEnabling := 1000 + nSeqEnabling;
		END_IF
		
		
	50: //Deside if or if not add enviroment to group
		IF XPlanarParameterlist.B_ADD_ENVIROMENT_TO_GROUP THEN
			nSeqEnabling := 51;
		ELSE
			nSeqEnabling := 70;
		END_IF
		
	51: // Add environment to group
		hr := ipEnvironment.AddToGroup(ipGroup);
		
		IF CheckOk(hr) THEN 
			nSeqEnabling := 52;
		ELSE
			nSeqEnabling := 1000 + nSeqEnabling;
		END_IF		

	52: // Adding environment to group
		hr := ipEnvironment.Feedback.HR;
		
		IF CheckOk(hr) THEN 
			nSeqEnabling := 70;
		ELSIF FAILED(hr) THEN
			nSeqEnabling := 1000 + nSeqEnabling;
		END_IF

		
	70: // Configure the tracks |
		THIS^.fbTracks.ResetIterator();
		WHILE THIS^.fbTracks.HasNextObject() DO
			IF ToXpTrack(THIS^.fbTracks.GetNextObject(),ipTempTrack) THEN
				hr := GetMostSignificant(hr, ipTempTrack.Configure());
			END_IF
		END_WHILE
		
		IF CheckOk(hr) THEN 
			nSeqEnabling := 71;
		ELSE
			nSeqEnabling := 1000 + nSeqEnabling;
		END_IF	
		
	71: // Configuring the tracks 
		THIS^.fbTracks.ResetIterator();
		WHILE THIS^.fbTracks.HasNextObject() DO
			IF ToXpTrack(THIS^.fbTracks.GetNextObject(),ipTempTrack) THEN
				hr := GetMostSignificant(hr, ipTempTrack.Configuring());
			END_IF
		END_WHILE
		
		IF CheckOk(hr) THEN 
			nSeqEnabling := 80;
		ELSIF FAILED(hr) THEN
			nSeqEnabling := 1000 + nSeqEnabling;
		END_IF	
		
		
	80: // Enable the tracks
		THIS^.fbTracks.ResetIterator();
		WHILE THIS^.fbTracks.HasNextObject() DO
			IF ToXpTrack(THIS^.fbTracks.GetNextObject(),ipTempTrack) THEN
				hr := GetMostSignificant(hr, ipTempTrack.Enable());
			END_IF
		END_WHILE
		
		IF CheckOk(hr) THEN 
			nSeqEnabling := 81;
		ELSE
			nSeqEnabling := 1000 + nSeqEnabling;
		END_IF		

	81: // Enabling the tracks
		THIS^.fbTracks.ResetIterator();
		WHILE THIS^.fbTracks.HasNextObject() DO
			IF ToXpTrack(THIS^.fbTracks.GetNextObject(),ipTempTrack) THEN
				hr := GetMostSignificant(hr, ipTempTrack.Feedback.HR);
			END_IF
		END_WHILE
		
		IF CheckOk(hr) THEN 
			nSeqEnabling := 90;
		ELSIF FAILED(hr) THEN
			nSeqEnabling := 1000 + nSeqEnabling;
		END_IF	
		
		
	90: // Add tracks to group
		THIS^.fbTracks.ResetIterator();
		WHILE THIS^.fbTracks.HasNextObject() DO
			IF ToXpTrack(THIS^.fbTracks.GetNextObject(),ipTempTrack) THEN
				hr := GetMostSignificant(hr, ipTempTrack.AddToGroup(ipGroup));
			END_IF
		END_WHILE
		
		IF CheckOk(hr) THEN 
			nSeqEnabling := 91;
		ELSE
			nSeqEnabling := 1000 + nSeqEnabling;
		END_IF	

	91: // Adding tracks to group
		THIS^.fbTracks.ResetIterator();
		WHILE THIS^.fbTracks.HasNextObject() DO
			IF ToXpTrack(THIS^.fbTracks.GetNextObject(),ipTempTrack) THEN
				hr := GetMostSignificant(hr, ipTempTrack.Feedback.HR);
			END_IF
		END_WHILE
		
		IF CheckOk(hr) THEN 
			nSeqEnabling := 100;
		ELSIF FAILED(hr) THEN
			nSeqEnabling := 1000 + nSeqEnabling;
		END_IF		
			
		
		
	100: // Config Station
		THIS^.fbStations.ResetIterator();
		WHILE THIS^.fbStations.HasNextObject() DO
			IF ToXpStation(THIS^.fbStations.GetNextObject(),ipTempStation) THEN
				hr := GetMostSignificant(hr, ipTempStation.Configure());
			END_IF
		END_WHILE
		
		IF CheckOk(hr) THEN 
			nSeqEnabling := 110;
		ELSE
			nSeqEnabling := 1000 + nSeqEnabling;
		END_IF

		
		
	110: // Enable movers
		THIS^.fbMovers.ResetIterator();
		WHILE THIS^.fbMovers.HasNextObject() DO
			IF ToXpMover(THIS^.fbMovers.GetNextObject(),ipTempMover) THEN
				hr := GetMostSignificant(hr, ipTempMover.Enable());
			END_IF
		END_WHILE
		
		IF CheckOk(hr) THEN 
			nSeqEnabling := 111;
		ELSE
			nSeqEnabling := 1000 + nSeqEnabling;
		END_IF	
		
	111: // Enabling movers
		THIS^.fbMovers.ResetIterator();
		WHILE THIS^.fbMovers.HasNextObject() DO
			IF ToXpMover(THIS^.fbMovers.GetNextObject(),ipTempMover) THEN
				hr := GetMostSignificant(hr, ipTempMover.Feedback.HR);
			END_IF
		END_WHILE
		
		IF CheckOk(hr) THEN 
			nSeqEnabling := 120;
		ELSIF FAILED(hr) THEN
			nSeqEnabling := 1000 + nSeqEnabling;
		END_IF	
		

	120: //Rotate A-Axis to zero
		THIS^.fbMovers.ResetIterator();
		WHILE THIS^.fbMovers.HasNextObject() DO
			IF ToXpMover(THIS^.fbMovers.GetNextObject(),ipTempMover) THEN
				hr := GetMostSignificant(hr, ipTempMover.MoveA(0));
			END_IF
		END_WHILE
		
		IF CheckOk(hr) THEN 
			nSeqEnabling := 121;
		ELSE
			nSeqEnabling := 1000 + nSeqEnabling;
		END_IF	
		
	121: //Rotating A-Axis to Zero			
		THIS^.fbMovers.ResetIterator();
		WHILE THIS^.fbMovers.HasNextObject() DO
			IF ToXpMover(THIS^.fbMovers.GetNextObject(),ipTempMover) THEN
				hr := GetMostSignificant(hr, ipTempMover.Feedback.HR);
			END_IF
		END_WHILE
		
		IF CheckOk(hr) THEN 
			nSeqEnabling := 122;
		ELSIF FAILED(hr) THEN
			nSeqEnabling := 1000 + nSeqEnabling;
		END_IF	
		
	122: //Rotate B-Axis to zero
		THIS^.fbMovers.ResetIterator();
		WHILE THIS^.fbMovers.HasNextObject() DO
			IF ToXpMover(THIS^.fbMovers.GetNextObject(),ipTempMover) THEN
				hr := GetMostSignificant(hr, ipTempMover.MoveB(0));
			END_IF
		END_WHILE
		
		IF CheckOk(hr) THEN 
			nSeqEnabling := 123;
		ELSE
			nSeqEnabling := 1000 + nSeqEnabling;
		END_IF	
		
	123: //Rotating B-Axis to zero			
		THIS^.fbMovers.ResetIterator();
		WHILE THIS^.fbMovers.HasNextObject() DO
			IF ToXpMover(THIS^.fbMovers.GetNextObject(),ipTempMover) THEN
				hr := GetMostSignificant(hr, ipTempMover.Feedback.HR);
			END_IF
		END_WHILE
		
		IF CheckOk(hr) THEN 
			nSeqEnabling := 130;
		ELSIF FAILED(hr) THEN
			nSeqEnabling := 1000 + nSeqEnabling;
		END_IF		
		
				
		
	130: //Rotate C-Axis to "Zero" (to the next 90 degree pitch)
		THIS^.fbMovers.ResetIterator();
		WHILE THIS^.fbMovers.HasNextObject() DO
			IF ToXpMover(THIS^.fbMovers.GetNextObject(),ipTempMover) THEN
				// Decide which 90 degree pitch is closer to the current position. If the remainder is greater than 45 degrees, then round up to the next 90 degree division.
				lrCRotationShortestPos := LREAL_TO_DINT(ipTempMover.PlanarMover.MCTOPLC.SET.SetPos.C / 90.0) * 90.0;
				hr := GetMostSignificant(hr, ipTempMover.MoveC(	fPosition		:= lrCRotationShortestPos, 
																additionalTurns := 0,
																direction		:= Tc3_Mc3Definitions.MC_DIRECTION.mcDirectionShortestWay));
			END_IF
		END_WHILE
		
		IF CheckOk(hr) THEN 
			nSeqEnabling := 131;
		ELSE
			nSeqEnabling := 1000 + nSeqEnabling;
		END_IF	
		
	131: //Rotating C-Axis to Zero			
		THIS^.fbMovers.ResetIterator();
		WHILE THIS^.fbMovers.HasNextObject() DO
			IF ToXpMover(THIS^.fbMovers.GetNextObject(),ipTempMover) THEN
				hr := GetMostSignificant(hr, ipTempMover.Feedback.HR);
			END_IF
		END_WHILE
		
		IF CheckOk(hr) THEN 
			nSeqEnabling := 140;
		ELSIF FAILED(hr) THEN
			nSeqEnabling := 1000 + nSeqEnabling;
		END_IF	
			
		
		
	140: // Add movers to group
		THIS^.fbMovers.ResetIterator();
		WHILE THIS^.fbMovers.HasNextObject() DO
			IF ToXpMover(THIS^.fbMovers.GetNextObject(),ipTempMover) THEN
				hr := GetMostSignificant(hr, ipTempMover.AddToGroup(THIS^.ipGroup));
			END_IF
		END_WHILE
		
		IF CheckOk(hr) THEN 
			nSeqEnabling := 141;
		ELSE
			nSeqEnabling := 1000 + nSeqEnabling;
		END_IF	
	
	141: // Adding mover to group
		THIS^.fbMovers.ResetIterator();
		WHILE THIS^.fbMovers.HasNextObject() DO
			IF ToXpMover(THIS^.fbMovers.GetNextObject(),ipTempMover) THEN
				hr := GetMostSignificant(hr, ipTempMover.Feedback.HR);
			END_IF
		END_WHILE
		
		IF CheckOk(hr) THEN 
			nSeqEnabling := 150;
		ELSIF FAILED(hr) THEN
			nSeqEnabling := 1000 + nSeqEnabling;
		END_IF		
	
		
		
	150: // Enable group
		hr := ipGroup.Enable();
		
		IF CheckOk(hr) THEN 
			nSeqEnabling := 151;
		ELSE
			nSeqEnabling := 1000 + nSeqEnabling;
		END_IF	
		
	151: // Enabling group
		hr := ipGroup.Feedback.HR;
		
		IF CheckOk(hr) THEN 
			nSeqEnabling := 190;
		ELSIF FAILED(hr) THEN
			nSeqEnabling := 1000 + nSeqEnabling;
		END_IF	

		
//	170: // Waiting movers are in free movement
//		THIS^.fbMovers.ResetIterator();
//		WHILE THIS^.fbMovers.HasNextObject() DO
//			IF ToXpMover(THIS^.fbMovers.GetNextObject(),ipTempMover) THEN
//				hr := GetMostSignificant(hr, ipTempMover.Feedback.HR);
//				IF NOT (ipTempMover.Mode = MC_PLANAR_MOVER_COMMAND_MODE.FreeMovement) THEN
//					hr := GetMostSignificant(hr, S_PENDING);
//				END_IF
//			END_IF
//		END_WHILE
//		
//		IF CheckOk(hr) THEN 
//			nSeqEnabling := 180;
//		ELSIF FAILED(hr) THEN
//			nSeqEnabling := 1000 + nSeqEnabling;
//		END_IF	
				
		
		
		
	190: (*	Restart of the sequenze "JoiningTrack". Default strategy is that each mover joins the closest track
			Outsourced to a method for easier overwriting *)
		THIS^.nSeqJoiningTrack := 0;	
		nSeqEnabling := 191;	

	191: (*	Default strategy is that each mover joins the closest track
			Outsourced to a method for easier overwriting *)
		hr := THIS^.JoiningTrack();

		IF CheckOk(hr) THEN 
			nSeqEnabling := 200;
		ELSIF FAILED(hr) THEN
			nSeqEnabling := 1000 + nSeqEnabling;
		END_IF	
		
	

	
	200: (*	Restart of the sequenze "JoiningStation" to distribute the movers to the available stations.
			Outsourced to a method for easier overwriting *)
		THIS^.nSeqJoiningStation := 0;	
		nSeqEnabling := 201;	
	
	201: (*	Distribute the movers to the available stations.
		 	Outsourced to a method for easier overwriting *)
		hr := THIS^.JoiningStation();

		IF CheckOk(hr) THEN 
			nSeqEnabling := SEQ_DONE;
		ELSIF FAILED(hr) THEN
			nSeqEnabling := 1000 + nSeqEnabling;
		END_IF	


		
		
	SEQ_DONE: // Done
		Enabling := S_OK;

		
	1000..1999://Error
		hr := GetMostSignificant(hr, E_FAIL);
END_CASE


//Timeout after to long stay in one of the following seq.
fbTimeOutSeq.IN := (nSeqEnabling = 5) AND (nlastState = nSeqEnabling);
fbTimeOutSeq.PT := T#5S;
fbTimeOutSeq();
nlastState := nSeqEnabling;


IF fbTimeOutSeq.Q THEN
	//next seq is error
	nSeqEnabling := 1000 + nSeqEnabling;
END_IF


// Propagate error
IF FAILED(hr) THEN
	Enabling := hr;
END_IF
END_METHOD

METHOD Initialize : HRESULT
VAR_INPUT
END_VAR
VAR
	hr 				: HRESULT := S_OK;
	ipEachStation 	: I_XP_Station;
END_VAR
THIS^.eActiveCommand 					:= CHALET_NC.E_NcAxisCommands.Initialize;
THIS^.fbFeedback.LastCommandAccepted	:= TRUE;		
THIS^.fbFeedback.Busy 					:= TRUE;

//Check Error during FB_Init
IF THIS^.bErrorDuringFbInit THEN
	Initialize:= E_FAIL;
	RETURN;
END_IF	


//Check if Envirement and Group is existing
IF THIS^.ipEnvironment = 0 OR THIS^.ipGroup = 0 THEN
	Initialize:= E_FAIL;
	RETURN;
END_IF	


//Init envirement first to get access to XTS_Utility
IF THIS^.ipEnvironment.Initialize() = S_OK THEN
	hr := GetMostSignificant(hr, THIS^.ipGroup.Initialize());
	hr := GetMostSignificant(hr, THIS^.fbMovers.Initialize());
	hr := GetMostSignificant(hr, THIS^.fbTracks.Initialize());
	hr := GetMostSignificant(hr, THIS^.fbStations.Initialize());
	hr := GetMostSignificant(hr, THIS^.fbTriggers.Initialize());
	hr := GetMostSignificant(hr, THIS^.fbZones.Initialize());
ELSE
	hr := S_PENDING;
END_IF	



THIS^.bInitDone := (hr = S_OK);

Initialize:= hr;

THIS^.fbFeedback.HR := Initialize;
END_METHOD

{attribute 'monitoring':='call'}
PROPERTY Initialized : BOOL
GET
Initialized := bInitDone;
END_GET
END_PROPERTY

METHOD Station : I_XP_Station_PLC
VAR_INPUT
	sLUID : STRING;
END_VAR
//IF no station was found, INTERFACE is 0 -> can generate fatal error
__QUERYINTERFACE(THIS^.fbStations.FindLUID(sLUID),Station);
END_METHOD

METHOD ValideStationGroupID : BOOL //Return TRUE if group is existing
VAR_INPUT
	sStationGroupID	: STRING; //Group of the targed station
END_VAR
VAR
	ipEachStation : I_XP_Station_PLC;
END_VAR
THIS^.fbStations.ResetIterator();
WHILE THIS^.fbStations.HasNextObject() DO
	IF __QUERYINTERFACE(THIS^.fbStations.GetNextObject(),ipEachStation) THEN
		//Return TRUE if found
		IF (ipEachStation.StationGroupID = sStationGroupID) THEN
			ValideStationGroupID := TRUE;
			RETURN;
		END_IF
	END_IF
END_WHILE
END_METHOD

//Return TRUE if unique station id is valid. if false, interfacepointer is zero -> fatal error
METHOD ValidLUID : BOOL
VAR_INPUT
	sLUID : STRING;
END_VAR
VAR
	ipStation : I_XP_Station_PLC;
END_VAR
ipStation := THIS^.Station(sLUID);
ValidLUID := (ipStation <> 0);
END_METHOD

METHOD LinkEnvironment : HRESULT
VAR_INPUT
	ipEnvironment : I_CH_Object;
END_VAR

VAR
	ipXpEnvironment : I_XP_Environment;
END_VAR
IF ipEnvironment <> 0 AND_THEN __QUERYINTERFACE(ipEnvironment,ipXpEnvironment) THEN
	THIS^.ipEnvironment := ipXpEnvironment;
ELSE
	LinkEnvironment := E_FAIL;
	THIS^.bErrorDuringFbInit := TRUE;
END_IF
END_METHOD

METHOD LinkGroup : HRESULT
VAR_INPUT
	ipGroup : I_CH_Object;
END_VAR

VAR
	ipXpGroup : I_XP_Group;
END_VAR
IF ipGroup <> 0 AND_THEN __QUERYINTERFACE(ipGroup,ipXpGroup) THEN
	THIS^.ipGroup := ipXpGroup;
ELSE
	LinkGroup := E_FAIL;
	THIS^.bErrorDuringFbInit := TRUE;
END_IF
END_METHOD

METHOD RegisterMover : HRESULT
VAR_INPUT
	ipMover : I_CH_Object;
END_VAR

VAR
	ipXpMover : I_XP_Mover;
END_VAR
IF ipMover = 0 THEN
	//Invalide interface	
	THIS^.bErrorDuringFbInit := TRUE;
	RegisterMover := E_FAIL;
	
ELSIF NOT __QUERYINTERFACE(ipMover, ipXpMover) THEN
	//The required interface is missing
	THIS^.bErrorDuringFbInit := TRUE;
	RegisterMover := E_FAIL;
	
ELSIF THIS^.fbMovers.IsFull THEN
	//List is full
	THIS^.bErrorDuringFbInit := TRUE;
	RegisterMover := E_FAIL;
	
ELSIF THIS^.bInitDone THEN
	//To late. System is initilized
	THIS^.bErrorDuringFbInit := TRUE;
	RegisterMover := E_FAIL;
	
ELSE
	
	THIS^.fbMovers.AddObject(ipMover);
END_IF
END_METHOD

METHOD RegisterStation : HRESULT
VAR_INPUT
	ipStation : I_CH_Object;
END_VAR

VAR
	ipXpStation : I_XP_Station;
END_VAR
IF ipStation = 0 THEN
	//Invalide interface	
	THIS^.bErrorDuringFbInit := TRUE;
	RegisterStation := E_FAIL;
	
ELSIF NOT __QUERYINTERFACE(ipStation, ipXpStation) THEN
	//The required interface is missing
	THIS^.bErrorDuringFbInit := TRUE;
	RegisterStation := E_FAIL;
	
ELSIF THIS^.fbStations.IsFull THEN
	//List is full
	THIS^.bErrorDuringFbInit := TRUE;
	RegisterStation := E_FAIL;
	
ELSIF THIS^.bInitDone THEN
	//To late. System is initilized
	THIS^.bErrorDuringFbInit := TRUE;
	RegisterStation := E_FAIL;
		
ELSE
	
	THIS^.fbStations.AddObject(ipStation);
END_IF
END_METHOD

METHOD RegisterTrack : HRESULT
VAR_INPUT
	ipTrack : I_CH_Object;
END_VAR

VAR
	ipXpTrack : I_XP_Track;
END_VAR
IF ipTrack = 0 THEN
	//Invalide interface	
	THIS^.bErrorDuringFbInit := TRUE;
	RegisterTrack := E_FAIL;
	
ELSIF NOT __QUERYINTERFACE(ipTrack, ipXpTrack) THEN
	//The required interface is missing
	THIS^.bErrorDuringFbInit := TRUE;
	RegisterTrack := E_FAIL;
	
ELSIF THIS^.fbTracks.IsFull THEN
	//List is full
	THIS^.bErrorDuringFbInit := TRUE;
	RegisterTrack := E_FAIL;
	
ELSIF THIS^.bInitDone THEN
	//To late. System is initilized
	THIS^.bErrorDuringFbInit := TRUE;
	RegisterTrack := E_FAIL;
		
ELSE
	
	THIS^.fbTracks.AddObject(ipTrack);
END_IF
END_METHOD

METHOD RegisterTrigger : HRESULT
VAR_INPUT
	ipTrigger	: CHALET_BaseComponents.I_CH_Object;
END_VAR
VAR
	ipXpTrigger : I_Xp_Trigger;
END_VAR
IF ipTrigger = 0 THEN
	//Invalide interface	
	THIS^.bErrorDuringFbInit := TRUE;
	RegisterTrigger := E_FAIL;
	
ELSIF NOT __QUERYINTERFACE(ipTrigger, ipXpTrigger) THEN
	//The required interface is missing
	THIS^.bErrorDuringFbInit := TRUE;
	RegisterTrigger := E_FAIL;
	
ELSIF THIS^.fbTriggers.IsFull THEN
	//List is full
	THIS^.bErrorDuringFbInit := TRUE;
	RegisterTrigger := E_FAIL;
	
ELSIF THIS^.bInitDone THEN
	//To late. System is initilized
	THIS^.bErrorDuringFbInit := TRUE;
	RegisterTrigger := E_FAIL;
		
ELSE
	
	THIS^.fbTriggers.AddObject(ipTrigger);
END_IF
END_METHOD

METHOD RegisterZone : HRESULT
VAR_INPUT
	ipZone	: CHALET_BaseComponents.I_CH_Object;
END_VAR
VAR
	ipXpsZone : I_XP_Zone;
END_VAR
IF ipZone = 0 THEN
	//Invalide interface	
	THIS^.bErrorDuringFbInit := TRUE;
	RegisterZone := E_FAIL;

ELSIF NOT __QUERYINTERFACE(ipZone, ipXpsZone) THEN
	//The required interface is missing
	THIS^.bErrorDuringFbInit := TRUE;
	RegisterZone := E_FAIL;
	
ELSIF THIS^.fbZones.IsFull THEN
	//List is full
	THIS^.bErrorDuringFbInit := TRUE;
	RegisterZone := E_FAIL;
	
ELSIF THIS^.bInitDone THEN
	//To late. System is initilized
	THIS^.bErrorDuringFbInit := TRUE;
	RegisterZone := E_FAIL;
		
ELSE
	
	THIS^.fbZones.AddObject(ipZone);	
END_IF
END_METHOD

{attribute 'monitoring':='call'}
PROPERTY Enviroment : I_XP_Environment
GET
Enviroment := THIS^.ipEnvironment;
END_GET
END_PROPERTY

{attribute 'monitoring':='call'}
PROPERTY Feedback : CHALET_BaseComponents.I_CH_Feedback
GET
Feedback := THIS^.fbFeedback;
END_GET
END_PROPERTY

{attribute 'monitoring':='call'}
PROPERTY Movers : CHALET_BaseComponents.I_CH_LIST
GET
Movers := THIS^.fbMovers;
END_GET
END_PROPERTY

{attribute 'monitoring':='call'}
PROPERTY Stations : CHALET_BaseComponents.I_CH_LIST
GET
Stations := THIS^.fbStations;
END_GET
END_PROPERTY

{attribute 'monitoring':='call'}
PROPERTY Tracks : CHALET_BaseComponents.I_CH_LIST
GET
Tracks := THIS^.fbTracks;
END_GET
END_PROPERTY

{attribute 'monitoring':='call'}
PROPERTY Triggers : CHALET_BaseComponents.I_CH_LIST
GET
Triggers := THIS^.fbTriggers;
END_GET
END_PROPERTY

METHOD Update : HRESULT
VAR_INPUT
END_VAR
VAR
	hr : HRESULT;
END_VAR
hr := S_OK;


hr := GetMostSignificant(hr, THIS^.Enabling());
hr := GetMostSignificant(hr, THIS^.Disabling());




// ********************** Set feedback depending on active command *******************************
IF THIS^.eActiveCommand <> E_NcAxisCommands.None THEN
	fbFeedback.ActiveCommand 	:= TO_STRING(THIS^.eActiveCommand);	
END_IF

CASE THIS^.eActiveCommand OF
	E_NcAxisCommands.None: 
		;

	E_NcAxisCommands.Initialize:
		fbFeedback.Busy 		:= NOT THIS^.bInitDone;
		fbFeedback.Done 		:= THIS^.bInitDone;
		fbFeedback.ErrorId 		:= 0;
		
	E_NcAxisCommands.Enable:
		fbFeedback.Busy 		:= nSeqEnabling > 0;
		fbFeedback.Done 		:= THIS^.Enabled;
		IF nSeqEnabling > 1000 THEN
			fbFeedback.ErrorId 		:= nSeqEnabling;
		END_IF
		
	E_NcAxisCommands.Disable:
		fbFeedback.Busy 		:= nSeqDisabling > 0;
		fbFeedback.Done 		:= THIS^.Disabled;
		IF nSeqDisabling > 1000 THEN
			fbFeedback.ErrorId 		:= nSeqDisabling;
		END_IF
		


	ELSE//External command in subclass
		;
END_CASE


// **********************  Stop to execute commands on .done or .error ***************************
IF fbFeedback.Done OR THIS^.fbFeedback.Error THEN
	eActiveCommand 				:= E_NcAxisCommands.None;
END_IF







hr := GetMostSignificant(hr, THIS^.fbMovers.Update());
hr := GetMostSignificant(hr, THIS^.fbTracks.Update());
hr := GetMostSignificant(hr, THIS^.fbStations.Update());
hr := GetMostSignificant(hr, THIS^.fbZones.Update());
hr := GetMostSignificant(hr, THIS^.fbTriggers.Update());
hr := GetMostSignificant(hr, THIS^.ipGroup.Update());
hr := GetMostSignificant(hr, THIS^.ipEnvironment.Update());


Update:= hr;
END_METHOD

{attribute 'monitoring':='call'}
PROPERTY Zones : CHALET_BaseComponents.I_CH_LIST
GET
Zones := THIS^.fbZones;
END_GET
END_PROPERTY

END_FUNCTION_BLOCK

// COMPONENTs/Track/FB_XP_Track
{attribute 'no_explicit_call' := 'Do not call the body - Stick to OOP'}
(* XPlanar track - n per associated XPlanar. Can be instantiated as an array and/or individually
	The Planar track is a software object that represents a (virtual) one-dimensional path on the two-dimensional XPlanar stator surface. 
	Several Planar movers can be lined up and moved on this path. Collisions are prevented by keeping a preset distance between the movers. *)	
FUNCTION_BLOCK FB_XP_Track EXTENDS FB_CH_Object IMPLEMENTS I_XP_Track
VAR
	//Link to Planar-Track object
	fbTrack : MC_PlanarTrack;
	
	{attribute 'hide'}  
	bInitDone :BOOL := FALSE;
	{attribute 'hide'}               	
	fbFeedback 			: FB_XP_Feedback;
	{attribute 'hide'}                   	
	eActiveCommand 		: CHALET_Nc.E_NcAxisCommands := CHALET_Nc.E_NcAxisCommands.None;
	{attribute 'hide'}
	ipXpSystem : I_XP_System_Registration;
	{attribute 'hide'}	
	nSeqConfiguring : UINT;
	{attribute 'hide'} 
	ipTracksEndAtThis : ARRAY[0..(XPlanarParameterlist.N_MAX_STATIONS_AHEAD_OR_BEHIND-1)] OF I_XP_Track;
	{attribute 'hide'} 
	ipTracksStartFromThis : ARRAY[0..(XPlanarParameterlist.N_MAX_STATIONS_AHEAD_OR_BEHIND-1)] OF I_XP_Track;
	//HMI - The track is divided into an array of coordinates to display the track course on a visualization
	afTrackPoints		: ARRAY[0..XplanarParameterlist.N_TRACE_POINTS] OF PositionXY;
	

	{attribute 'hide'}
	// ipXpSystem Is Not Valid at this point, call the konstruktor again in the FB_Init
	fbSortedListMoversOnTrack	: FB_XP_Zone(ipXpSystem);
END_VAR

// Planar-Feedback objects
VAR
	{attribute 'hide'} 
	fbFeedbackDisable: MC_PlanarFeedback;
	{attribute 'hide'} 
	fbFeedbackEnable : MC_PlanarFeedback;
	{attribute 'hide'} 
	fbFeedbackAddToGrp : MC_PlanarFeedback;
	{attribute 'hide'} 
	fbFeedbackRmvFromGrp : MC_PlanarFeedback;
	{attribute 'hide'} 
	fbFeedbackReset : MC_PlanarFeedback;
END_VAR

METHOD Configure : HRESULT // This is called once during system enabling
VAR_INPUT
END_VAR
// Validate settings
IF THIS^.Length = 0 THEN
	Configure := E_FAIL;
	THIS^.fbFeedback.LastCommandAccepted:= FALSE;	
	RETURN;
END_IF

THIS^.eActiveCommand 				:= CHALET_NC.E_NcAxisCommands.Configure;
THIS^.fbFeedback.LastCommandAccepted:= TRUE;		
THIS^.fbFeedback.Busy 				:= TRUE;

THIS^.nSeqConfiguring := 10;
Configure := S_OK;
END_METHOD

METHOD Configuring : HRESULT // This is called until S_OK during system enabling
VAR
	ipEachTrackObj : I_CH_Object;
	nIdx : UDINT;
END_VAR
VAR_INST
	fbAdsRead 	: ADSREAD;
	TrackOTCID 	: ARRAY[0..(XPlanarParameterlist.N_MAX_STATIONS_AHEAD_OR_BEHIND-1)] OF OTCID;
END_VAR
VAR CONSTANT
	N_IDX_OFFSET_PREVIOUS_TRACK 	: UDINT := 16#050300D5; // Parameter(online) in Planar Track object
	N_IDX_OFFSET_SUBSEQUENT_TRACK 	: UDINT := 16#050300D6; // Parameter(online) in Planar Track object	
	
	N_PORT_MET_TASK 				: UINT := 521; //ZZZ TODO this port is not fix. REad from the TcCom object
END_VAR
Configuring := S_PENDING;
CASE nSeqConfiguring OF
	0: // Idle
		Configuring := S_OK;
		
	10: //Start
		//No config is done here. Set Track elements direkt in the Track TcCom Object
		nSeqConfiguring := 700;
		
	700: //Calculate an array of track points. These can then be visualized on an HMI, for example
		THIS^.CalcTrackPoints();
		nSeqConfiguring := 800;
	
	
	
	//PREVIOUS_TRACK
	800: // Prepare - Read from Track object
		fbAdsRead.READ := FALSE;
		MEMSET(destAddr := ADR(TrackOTCID), n := SIZEOF(TrackOTCID), fillByte:= 0);
		nSeqConfiguring := 801;
	
	801: // Start read - Read from Track object
		fbAdsRead.PORT		:= N_PORT_MET_TASK; 
		fbAdsRead.IDXGRP	:= THIS^.OID;
		fbAdsRead.IDXOFFS	:= N_IDX_OFFSET_PREVIOUS_TRACK; 
		fbAdsRead.LEN		:= SIZEOF(TrackOTCID);
		fbAdsRead.DESTADDR	:= ADR(TrackOTCID);
			
		fbAdsRead.READ := TRUE;
		nSeqConfiguring := 802;
	
	802: // Wait for reading - Read from Track object
		IF fbAdsRead.ERR AND fbAdsRead.ERRID = 6 THEN
			//Error, the reason for this could be that this track has no connected tracks
			//Continous with SUBSEQUENT_TRACK
			nSeqConfiguring := 850;
		ELSIF fbAdsRead.ERR THEN
			//Error
			nSeqConfiguring := nSeqConfiguring + 1000;
		ELSIF NOT fbAdsRead.BUSY THEN
			//Done
			nSeqConfiguring := 803;
		END_IF
	
	803: // Convert to I_XP_Track - Read from Track object
		FOR nIdx := 0 TO (XPlanarParameterlist.N_MAX_STATIONS_AHEAD_OR_BEHIND-1) DO
			//Get Obj
			ipEachTrackObj := THIS^.ipXpSystem.Tracks.FindOID(TrackOTCID[nIdx]);
			//convert obj -> I_XP_Track
			ToXpTrack(ipEachTrackObj, ipTracksEndAtThis[nIdx]);	
		END_FOR
		nSeqConfiguring := 850;		
	
		
		
		
	//SUBSEQUENT_TRACK	
	850: // Prepare - Read from Track object
		fbAdsRead.READ := FALSE;
		MEMSET(destAddr := ADR(TrackOTCID), n := SIZEOF(TrackOTCID), fillByte:= 0);
		nSeqConfiguring := 851;
	
	851: // Start read - Read from Track object
		fbAdsRead.PORT		:= N_PORT_MET_TASK;
		fbAdsRead.IDXGRP	:= THIS^.OID;
		fbAdsRead.IDXOFFS	:= N_IDX_OFFSET_SUBSEQUENT_TRACK;
		fbAdsRead.LEN		:= SIZEOF(TrackOTCID);
		fbAdsRead.DESTADDR	:= ADR(TrackOTCID);
			
		fbAdsRead.READ := TRUE;
		nSeqConfiguring := 852;
	
	852: // Wait for reading - Read from Track object
		IF fbAdsRead.ERR AND fbAdsRead.ERRID = 6 THEN
			//Error, the reason for this could be that this track has no connected tracks
			nSeqConfiguring := 900;
		ELSIF fbAdsRead.ERR THEN
			//Error
			nSeqConfiguring := nSeqConfiguring + 1000;
		ELSIF NOT fbAdsRead.BUSY THEN
			//Done
			nSeqConfiguring := 853;
		END_IF
	
	853: // Convert to I_XP_Track - Read from Track object
		FOR nIdx := 0 TO (XPlanarParameterlist.N_MAX_STATIONS_AHEAD_OR_BEHIND-1) DO
			//Get Obj
			ipEachTrackObj := THIS^.ipXpSystem.Tracks.FindOID(TrackOTCID[nIdx]);
			//convert obj -> I_XP_Track
			ToXpTrack(ipEachTrackObj, ipTracksStartFromThis[nIdx]);	
		END_FOR
		nSeqConfiguring := 900;
	
	
		
	
	
	900: // Config the internal FB_Zone
		THIS^.fbSortedListMoversOnTrack.AccocietedTrack 		:= (THIS^);
		THIS^.fbSortedListMoversOnTrack.StartPositionOnTrack	:= 0;
		THIS^.fbSortedListMoversOnTrack.EndPositionOnTrack 		:= THIS^.Length;
		nSeqConfiguring := 999;
		
	999: // Done
		Configuring := S_OK;
		
	1000..1999://Error
		Configuring := E_FAIL;
END_CASE


fbAdsRead();
END_METHOD

METHOD Disable : HRESULT
VAR_INPUT
END_VAR
IF NOT THIS^.fbFeedback.Busy THEN
	THIS^.eActiveCommand 				:= CHALET_NC.E_NcAxisCommands.Disable;
	THIS^.fbFeedback.LastCommandAccepted:= TRUE;		
	THIS^.fbFeedback.Busy 				:= TRUE;

	THIS^.fbTrack.Enable(fbFeedbackDisable);
	Disable := S_OK;
ELSE
	Disable := S_FALSE;
	THIS^.fbFeedback.LastCommandAccepted:= FALSE;	
END_IF
END_METHOD

METHOD Enable : HRESULT
VAR_INPUT
END_VAR
IF NOT THIS^.fbFeedback.Busy THEN
	THIS^.eActiveCommand 				:= CHALET_NC.E_NcAxisCommands.Enable;
	THIS^.fbFeedback.LastCommandAccepted:= TRUE;		
	THIS^.fbFeedback.Busy 				:= TRUE;

	THIS^.fbTrack.Enable(fbFeedbackEnable);
	Enable := S_OK;
ELSE
	Enable := S_FALSE;
	THIS^.fbFeedback.LastCommandAccepted:= FALSE;	
END_IF
END_METHOD

METHOD AddToGroup : HRESULT
VAR_INPUT
	iGroup : I_XP_Group;
END_VAR
IF NOT THIS^.fbFeedback.Busy THEN
	THIS^.eActiveCommand 				:= CHALET_NC.E_NcAxisCommands.AddToGroupe;
	THIS^.fbFeedback.LastCommandAccepted:= TRUE;		
	THIS^.fbFeedback.Busy 				:= TRUE;
	
	iGroup.AddTrack(THIS^.fbTrack, THIS^.fbFeedbackAddToGrp);
	AddToGroup := S_OK;
ELSE
	AddToGroup := S_FALSE;
	THIS^.fbFeedback.LastCommandAccepted:= FALSE;	
END_IF
END_METHOD

METHOD RemoveFromGroup : HRESULT
IF NOT THIS^.fbFeedback.Busy THEN
	THIS^.eActiveCommand 				:= CHALET_NC.E_NcAxisCommands.RemoveFromGroupe;
	THIS^.fbFeedback.LastCommandAccepted:= TRUE;		
	THIS^.fbFeedback.Busy 				:= TRUE;
	
	THIS^.fbTrack.RemoveFromGroup(THIS^.fbFeedbackRmvFromGrp);
	
	RemoveFromGroup := S_OK;
ELSE
	RemoveFromGroup := S_FALSE;
	THIS^.fbFeedback.LastCommandAccepted:= FALSE;	
END_IF
END_METHOD

METHOD AddMover : HRESULT
VAR_INPUT
	ipMover : I_XP_Mover;
END_VAR
IF ipMover <> 0 THEN
	AddMover := ipMover.JoinTrack(THIS^);
ELSE
	AddMover := E_FAIL;
END_IF
END_METHOD

METHOD PROTECTED CalcTrackPoints : HRESULT
VAR_INPUT
END_VAR
VAR
    nIdx      : UINT;
    fbPosition : PositionXYC;
	fLength   : LREAL;
END_VAR
fLength := THIS^.fbTrack.GetLength();

FOR nIdx := 0 TO XplanarParameterlist.N_TRACE_POINTS DO
	THIS^.fbTrack.GetPositionAt(fLength/(XplanarParameterlist.N_TRACE_POINTS)*nIdx, fbPosition);
	
	THIS^.afTrackPoints[nIdx].x := fbPosition.x;
	THIS^.afTrackPoints[nIdx].y := fbPosition.y;
	//THIS^.afTrackPoints[nIdx].c := fbPosition.c;
END_FOR

CalcTrackPoints := S_OK;
END_METHOD

{attribute 'monitoring':='call'}
PROPERTY CtsMoversOnTrack : UINT
GET
CtsMoversOnTrack := THIS^.fbSortedListMoversOnTrack.CtsMoversInZone;
END_GET
END_PROPERTY

METHOD FB_init : BOOL
VAR_INPUT
	bInitRetains : BOOL; // if TRUE, the retain variables are initialized (warm start / cold start)
	bInCopyCode : BOOL;  // if TRUE, the instance afterwards gets moved into the copy code (online change)
	
	ipSystem : I_CH_Object;
END_VAR
VAR_INST
	{attribute 'hide'}
	bFBInitCalledOnce : BOOL; //Do the following code once during start up and not during onlinechange
END_VAR
//Do the following code once during start up and not during onlinechange
IF NOT bFBInitCalledOnce THEN 
	
	(* Register to the Xplanar System
	   1. Test if the interface exists
	   2. Test if the object implements a "System for Mover" interface 
	*)
	IF ipSystem <> 0 AND_THEN __QUERYINTERFACE(ipSystem,THIS^.ipXpSystem) THEN
		THIS^.ipXpSystem.RegisterTrack(THIS^);
	END_IF
	
	THIS^.fbSortedListMoversOnTrack.FB_init(FALSE,FALSE, THIS^.ipXpSystem);
END_IF

bFBInitCalledOnce := TRUE;
END_METHOD

{attribute 'monitoring':='call'}
PROPERTY Feedback : I_XP_Feedback
GET
Feedback := THIS^.fbFeedback;
END_GET
END_PROPERTY

METHOD Initialize : HRESULT
VAR
	hr : HRESULT;
END_VAR
IF NOT THIS^.Mapped THEN
	//Error
	Initialize := E_FAIL;

ELSIF NOT bInitDone THEN
	//Busy
	Initialize := S_PENDING;
	
	//Config the internal FB_Zone
	THIS^.fbSortedListMoversOnTrack.AccocietedTrack 		:= (THIS^);
	THIS^.fbSortedListMoversOnTrack.StartPositionOnTrack	:= 0;
	THIS^.fbSortedListMoversOnTrack.EndPositionOnTrack 		:= 0; //End should be the length of track. But is not sure defind at this point
	THIS^.fbSortedListMoversOnTrack.ListOfMoversToCheck 	:= THIS^.ipXpSystem.Movers; // All Movers in system
	
	//Done as sone list is initilized
	bInitDone := (S_OK = THIS^.fbSortedListMoversOnTrack.Initialize());
	
ELSE	
	//Done
	Initialize := S_OK;	
END_IF



THIS^.fbFeedback.ActiveCommand 		:= TO_STRING(CHALET_NC.E_NcAxisCommands.Initialize);
THIS^.eActiveCommand 				:= CHALET_NC.E_NcAxisCommands.Initialize;
THIS^.fbFeedback.LastCommandAccepted:= TRUE;	
//Set done or keep in busy state	
THIS^.fbFeedback.HR := Initialize;
END_METHOD

{attribute 'monitoring':='call'}
PROPERTY Length : LREAL
GET
Length := THIS^.fbTrack.GetLength();
END_GET
END_PROPERTY

{attribute 'monitoring':='call'}
PROPERTY Mapped : BOOL //Project is mapped to MC (McToPlc and PlcToMc)
GET
VAR
	bMcToPlcNotMapped 	: BOOL;
END_VAR
bMcToPlcNotMapped := F_GetMappingStatus(ADR(THIS^.fbTrack.MCTOPLC_STD), SIZEOF(THIS^.fbTrack.MCTOPLC_STD)) <> EPlcMappingStatus.MS_Mapped;

Mapped := NOT bMcToPlcNotMapped;
END_GET
END_PROPERTY

{attribute 'monitoring':='call'}
PROPERTY MoversOnTrack : REFERENCE TO ARRAY [0..(CHALET_BaseComponents.BaseParameterlist.MAX_OBJECTS-1)] OF I_XP_Mover_PLC // Return a sorted list of movers on track. Index 0 is the mover in Front
GET
MoversOnTrack REF= THIS^.fbSortedListMoversOnTrack.MoversInZone;
END_GET
END_PROPERTY

{attribute 'monitoring':='call'}
PROPERTY OID : OTCID
GET
OID := THIS^.fbTrack.MCTOPLC_STD.TrackOID;
END_GET
END_PROPERTY

{attribute 'monitoring':='call'}
PROPERTY PlanarTrack : REFERENCE TO MC_PlanarTrack
GET
PlanarTrack ref= THIS^.fbTrack;
END_GET
END_PROPERTY

METHOD Reset : HRESULT
VAR_INPUT
END_VAR
THIS^.eActiveCommand 				:= CHALET_NC.E_NcAxisCommands.Reset;
THIS^.fbFeedback.LastCommandAccepted:= TRUE;		
THIS^.fbFeedback.Busy 				:= TRUE;

THIS^.fbTrack.Reset(THIS^.fbFeedbackReset);
Reset := S_OK;
END_METHOD

{attribute 'monitoring':='call'}
PROPERTY TracksEndAtThis : REFERENCE TO  ARRAY[0..(XPlanarParameterlist.N_MAX_STATIONS_AHEAD_OR_BEHIND-1)] OF I_XP_Track
GET
TracksEndAtThis REF= ipTracksEndAtThis;
END_GET
END_PROPERTY

{attribute 'monitoring':='call'}
PROPERTY TracksStartFromThis : REFERENCE TO ARRAY[0..(XPlanarParameterlist.N_MAX_STATIONS_AHEAD_OR_BEHIND-1)] OF I_XP_Track
GET
TracksStartFromThis REF= ipTracksStartFromThis;
END_GET
END_PROPERTY

METHOD PUBLIC Update : HRESULT
VAR_INPUT
END_VAR



// ********************** Set feedback depending on active command *******************************
IF THIS^.eActiveCommand <> E_NcAxisCommands.None THEN
	fbFeedback.ActiveCommand 	:= TO_STRING(THIS^.eActiveCommand);	
END_IF

CASE THIS^.eActiveCommand OF
	E_NcAxisCommands.None: 
		//Display if a Mover Error is active during no command is active
		IF THIS^.fbTrack.Error AND NOT fbFeedback.Error THEN 
			fbFeedback.ErrorId 			:= THIS^.fbTrack.ErrorID;
			fbFeedback.ActiveCommand 	:= TO_STRING(E_NcAxisCommands.None);	
			fbFeedback.ClearObjectInfo();
		END_IF

	E_NcAxisCommands.Initialize:
		fbFeedback.Busy 			:= NOT THIS^.bInitDone;
		fbFeedback.Done 			:= THIS^.bInitDone;
		fbFeedback.ErrorId 			:= 0;
		fbFeedback.ClearObjectInfo();
		                        	
	E_NcAxisCommands.Enable:     	
		fbFeedback.Busy 			:= fbFeedbackEnable.Busy;
		fbFeedback.Done 			:= fbFeedbackEnable.Done;
		fbFeedback.ErrorId 			:= fbFeedbackEnable.ErrorID;
        fbFeedback.ObjectInfo		:= fbFeedbackEnable.objectInfo;
                                			                        	
	E_NcAxisCommands.Disable:     	
		fbFeedback.Busy 			:= fbFeedbackDisable.Busy;
		fbFeedback.Done 			:= fbFeedbackDisable.Done;
		fbFeedback.ErrorId 			:= fbFeedbackDisable.ErrorID;
        fbFeedback.ObjectInfo		:= fbFeedbackDisable.objectInfo;
		
	E_NcAxisCommands.Configure:
		fbFeedback.Busy 		:= nSeqConfiguring > 0;
		fbFeedback.Done 		:= nSeqConfiguring = 999;
		IF nSeqConfiguring > 1000 THEN
			fbFeedback.ErrorId 		:= nSeqConfiguring;
		END_IF
                                			                        	
	E_NcAxisCommands.Reset:     	
		fbFeedback.Busy 			:= fbFeedbackReset.Busy;
		fbFeedback.Done 			:= fbFeedbackReset.Done;
		fbFeedback.ErrorId 			:= fbFeedbackReset.ErrorID;
        fbFeedback.ObjectInfo		:= fbFeedbackReset.objectInfo;
                                      			                        	
	E_NcAxisCommands.AddToGroupe:     	
		fbFeedback.Busy 			:= fbFeedbackAddToGrp.Busy;
		fbFeedback.Done 			:= fbFeedbackAddToGrp.Done;
		fbFeedback.ErrorId 			:= fbFeedbackAddToGrp.ErrorID;
        fbFeedback.ObjectInfo		:= fbFeedbackAddToGrp.objectInfo;
                                      			                        	
	E_NcAxisCommands.RemoveFromGroupe:     	
		fbFeedback.Busy 			:= fbFeedbackRmvFromGrp.Busy;
		fbFeedback.Done 			:= fbFeedbackRmvFromGrp.Done;
		fbFeedback.ErrorId 			:= fbFeedbackRmvFromGrp.ErrorID;
        fbFeedback.ObjectInfo		:= fbFeedbackRmvFromGrp.objectInfo;
                                		
	ELSE//External command in subclass
		;
END_CASE


// **********************  Stop to execute commands on .done or .error ***************************
IF fbFeedback.Done OR THIS^.fbFeedback.Error THEN
	eActiveCommand 				:= E_NcAxisCommands.None;
END_IF

//Update xplanar object
THIS^.fbTrack.Update();

//Update feedback object
fbFeedbackEnable.Update(); 
fbFeedbackDisable.Update(); 
fbFeedbackReset.Update(); 
fbFeedbackAddToGrp.Update(); 
fbFeedbackRmvFromGrp.Update();
END_METHOD

END_FUNCTION_BLOCK

// COMPONENTs/Track/I_XP_Track_PLC
INTERFACE I_XP_Track_PLC EXTENDS __SYSTEM.IQueryInterface

{attribute 'monitoring':='call'}
PROPERTY CtsMoversOnTrack : UINT
GET
END_GET
END_PROPERTY

{attribute 'monitoring':='call'}
PROPERTY Feedback : I_XP_Feedback
GET
END_GET
END_PROPERTY

{attribute 'monitoring':='call'}
PROPERTY Length : LREAL
GET
END_GET
END_PROPERTY

{attribute 'monitoring':='call'}
PROPERTY Mapped : BOOL //Project is mapped to MC (McToPlc and PlcToMc)
GET
END_GET
END_PROPERTY

{attribute 'monitoring':='call'}
PROPERTY MoversOnTrack : REFERENCE TO ARRAY [0..(CHALET_BaseComponents.BaseParameterlist.MAX_OBJECTS-1)] OF I_XP_Mover_PLC // Return a sorted list of movers on track. Index 0 is the mover in Front
GET
END_GET
END_PROPERTY

{attribute 'monitoring':='call'}
PROPERTY OID : OTCID
GET
END_GET
END_PROPERTY

{attribute 'monitoring':='call'}
PROPERTY PlanarTrack : REFERENCE TO MC_PlanarTrack
GET
END_GET
END_PROPERTY

{attribute 'monitoring':='call'}
PROPERTY TracksEndAtThis : REFERENCE TO  ARRAY[0..(XPlanarParameterlist.N_MAX_STATIONS_AHEAD_OR_BEHIND-1)] OF I_XP_Track
GET
END_GET
END_PROPERTY

{attribute 'monitoring':='call'}
PROPERTY TracksStartFromThis : REFERENCE TO ARRAY[0..(XPlanarParameterlist.N_MAX_STATIONS_AHEAD_OR_BEHIND-1)] OF I_XP_Track
GET
END_GET
END_PROPERTY

END_INTERFACE

// COMPONENTs/FUN_GetDistToPosModulo
FUNCTION FUN_GetDistToPosModulo : LREAL //This is only working in Positiv Direktion
VAR_INPUT
	fTargedPosition : LREAL;
	fActualPosition : LREAL;
	fModulo 		: LREAL;
END_VAR

VAR

END_VAR

IF fTargedPosition < fActualPosition THEN
	fTargedPosition := fTargedPosition + fModulo;
END_IF

FUN_GetDistToPosModulo := fTargedPosition - fActualPosition;

END_FUNCTION

// COMPONENTs/FUN_InLimitTest
FUNCTION FUN_InLimitTest : BOOL
VAR_INPUT
	fMinimum 	: LREAL;
	fMaximum 	: LREAL;
	fInput 		: LREAL;
END_VAR

//Normal case
// 9 Max
// 5 Test
// 1 Min
IF fMinimum <= fMaximum THEN
	FUN_InLimitTest := (fInput >= fMinimum) AND (fInput <= fMaximum);
	
//Modulo case	
// 6 | 6  Max
// 5 | 9  Test
// 8 | 8  Min
ELSIF fMinimum > fMaximum THEN
	FUN_InLimitTest := NOT((fInput > fMaximum) AND (fInput < fMinimum));
END_IF

END_FUNCTION
